// =============================================================================
// Version_Recipe - 06_MainProcess.scl
// Main process with recipe-based G-code and pre-scan validation
// =============================================================================

// -----------------------------------------------------------------------------
// FB_InputManager - OR-combine inputs from HMI, Panel, Remote
// DOC:
//  purpose: Create single rising-edge command outputs (Cmd_*) from multiple input sources.
//  inputs: HMI_*, Panel_*, Rem_* (Bool) - raw button states (level)
//  outputs: Cmd_* (Bool) - one-shot rising-edge commands for the system
//  notes: Uses prev* latches to detect rising edges; keeps logic simple for deterministic behavior.
// -----------------------------------------------------------------------------
FUNCTION_BLOCK "FB_InputManager"
{ S7_Optimized_Access := 'TRUE' }
VERSION : 1.0
    VAR_INPUT
        // Raw level inputs from various sources (HMI, physical panel, remote)
        HMI_Start : Bool;    // HMI Start button (level)
        HMI_Stop : Bool;     // HMI Stop button (level)
        HMI_Pause : Bool;    // HMI Pause button (level)
        HMI_Reset : Bool;    // HMI Reset button (level)
        Panel_Start : Bool;  // Physical panel Start
        Panel_Stop : Bool;   // Physical panel Stop
        Panel_Pause : Bool;  // Physical panel Pause
        Panel_Reset : Bool;  // Physical panel Reset
        Rem_Start : Bool;    // Remote Start (e.g. PLC network)
        Rem_Stop : Bool;     // Remote Stop
    END_VAR
    VAR_OUTPUT
        // One-shot command outputs (rising edge true for one cycle)
        Cmd_Start : Bool;
        Cmd_Stop : Bool;
        Cmd_Pause : Bool;
        Cmd_Reset : Bool;
    END_VAR
    VAR
        // Previous sampled raw values for edge detection
        prevStart : Bool;
        prevStop : Bool;
        prevPause : Bool;
        prevReset : Bool;
        // Combined raw inputs for current cycle
        rawStart : Bool;
        rawStop : Bool;
        rawPause : Bool;
        rawReset : Bool;
    END_VAR
BEGIN
    #rawStart := #HMI_Start OR #Panel_Start OR #Rem_Start;
    #rawStop := #HMI_Stop OR #Panel_Stop OR #Rem_Stop;
    #rawPause := #HMI_Pause OR #Panel_Pause;
    #rawReset := #HMI_Reset OR #Panel_Reset;
    #Cmd_Start := #rawStart AND NOT #prevStart;
    #Cmd_Stop := #rawStop AND NOT #prevStop;
    #Cmd_Pause := #rawPause AND NOT #prevPause;
    #Cmd_Reset := #rawReset AND NOT #prevReset;
    #prevStart := #rawStart; #prevStop := #rawStop; #prevPause := #rawPause; #prevReset := #rawReset;
END_FUNCTION_BLOCK

// -----------------------------------------------------------------------------
// FB_SafetyMonitor - Check E-Stop, Door, Air Pressure, Drives
// DOC:
//  purpose: Evaluate hardware safety inputs and bypass flags, produce SafeToRun/SafeToJog.
//  inputs: EStop_OK, Door_Closed, AirPressure_OK, DrivesReady and bypass flags.
//  outputs: SafeToRun (machine may start), SafeToJog (manual jog allowed), ErrorCode (if unsafe).
//  notes: Returns immediately on first fatal safety failure to minimize decision latency.
// -----------------------------------------------------------------------------
FUNCTION_BLOCK "FB_SafetyMonitor"
{ S7_Optimized_Access := 'TRUE' }
VERSION : 1.0
    VAR_INPUT
        EStop_OK : Bool;            // TRUE if E-stop circuit is OK (no emergency)
        Door_Closed : Bool;         // TRUE if safety door closed
        AirPressure_OK : Bool;      // TRUE if air pressure sufficient
        DrivesReady : Bool;         // TRUE if drives report ready
        // Bypass flags (from HMI) used only for testing; production should disable
        Bypass_EStop : Bool;
        Bypass_Door : Bool;
        Bypass_AirPressure : Bool;
        Bypass_Drives : Bool;
    END_VAR
    VAR_OUTPUT
        SafeToRun : Bool;           // TRUE => allowed to start program execution
        SafeToJog : Bool;           // TRUE => manual jogging permitted
        ErrorCode : Word;           // Non-zero if unsafe (map to DB_ErrorCodes)
    END_VAR
BEGIN
    // Runs every scan. RETURNs on first failing condition -- priority order matters.
    // EStop and Drive fault disable both SafeToRun and SafeToJog (jogging also forbidden).
    // Door and air pressure only disable SafeToRun (manual jog still permitted).
    #ErrorCode := 0;
    IF NOT #EStop_OK AND NOT #Bypass_EStop THEN
        // EMERGENCY STOP active -- all motion forbidden
        #SafeToRun := FALSE; #SafeToJog := FALSE; #ErrorCode := 16#0401;
        "DB_Diagnostic".Error_Text := 'Safety: EMERGENCY STOP active';
        RETURN;
    END_IF;
    // Drive readiness is NOT checked here.
    // In STATE_STOPPED, contactors are physically blocked (modePermit=0), so drives can never
    // report ready before starting. Blocking SafeToRun/SafeToJog here creates a deadlock.
    // Drive enable is handled automatically in STATE_STARTING (tonDriveReady timeout).
    // Drive faults while running are caught by prevDriveFaultX/Z detection → STATE_ERROR.
    #SafeToJog := TRUE;
    IF NOT #Door_Closed AND NOT #Bypass_Door THEN
        // Safety door open -- auto run forbidden, manual jog allowed
        #SafeToRun := FALSE; #ErrorCode := 16#0402;
        "DB_Diagnostic".Error_Text := 'Safety: Safety door is open';
        RETURN;
    END_IF;
    IF NOT #AirPressure_OK AND NOT #Bypass_AirPressure THEN
        // Air pressure insufficient -- pneumatic system will not operate
        #SafeToRun := FALSE; #ErrorCode := 16#0404;
        "DB_Diagnostic".Error_Text := 'Safety: Air pressure too low';
        RETURN;
    END_IF;
    #SafeToRun := TRUE;
END_FUNCTION_BLOCK

// -----------------------------------------------------------------------------
// FB_LimitMonitor - Check soft and hard limits
// DOC:
//  purpose: Validate current axis positions against configured soft limits and hardware limit switches.
//  inputs: ActualPos_X/Z, Homed_X/Z, HW limit switches.
//  outputs: LimitError (TRUE if any violation), ErrorCode (first matching error code).
//  notes: Soft limits from DB_MachineConfig are used; hardware limit switches take precedence.
//         Soft limits are only checked for a HOMED axis (Homed_X/Z = StatusBits.HomingDone):
//         before homing the TO position is meaningless (0 after restart, stale after a run),
//         so comparing it against limits would produce false trips.
// -----------------------------------------------------------------------------
FUNCTION_BLOCK "FB_LimitMonitor"
{ S7_Optimized_Access := 'TRUE' }
VERSION : 1.0
    VAR_INPUT
        ActualPos_X : Real;         // Current X position (mm)
        ActualPos_Z : Real;         // Current Z position (mm)
        Homed_X : Bool;             // X axis homed (StatusBits.HomingDone) -- soft limits checked only when TRUE
        Homed_Z : Bool;             // Z axis homed (StatusBits.HomingDone) -- soft limits checked only when TRUE
        // NC limit switches: TRUE=closed=OK, FALSE=open=limit triggered
        // Cable break also reads FALSE → fail-safe behavior
        HW_NC_X_Min : Bool;         // NC switch: X min (FALSE = limit hit)
        HW_NC_X_Max : Bool;         // NC switch: X max (FALSE = limit hit)
        HW_NC_Z_Min : Bool;         // NC switch: Z min (FALSE = limit hit)
        HW_NC_Z_Max : Bool;         // NC switch: Z max (FALSE = limit hit)
        // PNP NO proximity sensors: TRUE=target detected=entered limit zone
        // Triggered BEFORE NC switch → early warning + second safety layer
        HW_PNP_X_Min : Bool;        // PNP NO sensor: X min (TRUE = limit zone)
        HW_PNP_X_Max : Bool;        // PNP NO sensor: X max (TRUE = limit zone)
        HW_PNP_Z_Min : Bool;        // PNP NO sensor: Z min (TRUE = limit zone)
        HW_PNP_Z_Max : Bool;        // PNP NO sensor: Z max (TRUE = limit zone)
    END_VAR
    VAR_OUTPUT
        LimitError : Bool;          // TRUE if any soft/hard limit violated
        ErrorCode : Word;           // Specific error code for HMI/alarm
    END_VAR
BEGIN
    // Runs every scan. Soft limits are read from DB_MachineConfig.
    // Hardware limit switches take priority over soft limits (physical end stop).
    // ErrorCode shows the last triggered fault -- multiple can be active simultaneously.
    #LimitError := FALSE; #ErrorCode := 0;
    // --- Software (Soft) Limits ---
    // Only checked while the axis is homed: an un-homed axis has no valid position
    // reference, so soft limits cannot mean anything before the reference seek completes.
    IF #Homed_X THEN
        IF #ActualPos_X < "DB_MachineConfig".SoftLimit_MinX THEN
            #LimitError := TRUE; #ErrorCode := 16#0101;
            "DB_Diagnostic".Error_Text := 'Limit: X axis below minimum soft limit';
        END_IF;
        IF #ActualPos_X > "DB_MachineConfig".SoftLimit_MaxX THEN
            #LimitError := TRUE; #ErrorCode := 16#0102;
            "DB_Diagnostic".Error_Text := 'Limit: X axis above maximum soft limit';
        END_IF;
    END_IF;
    IF #Homed_Z THEN
        IF #ActualPos_Z < "DB_MachineConfig".SoftLimit_MinZ THEN
            #LimitError := TRUE; #ErrorCode := 16#0103;
            "DB_Diagnostic".Error_Text := 'Limit: Z axis below minimum soft limit';
        END_IF;
        IF #ActualPos_Z > "DB_MachineConfig".SoftLimit_MaxZ THEN
            #LimitError := TRUE; #ErrorCode := 16#0104;
            "DB_Diagnostic".Error_Text := 'Limit: Z axis above maximum soft limit';
        END_IF;
    END_IF;
    // --- Hardware Limit Switches ---
    // NC switches: the TO (Technology Object) is configured with these as HW limits.
    // The TO handles deceleration and stop directly -- no PLC action required.
    // Only E-Stop cuts contactor power; PLC does NOT raise LimitError on NC hits.
    //
    // PNP proximity sensors: handled separately in FB_Process (inline halt block).
    // In auto mode: PNP → MC_Halt on triggered axis + STATE_ERROR (codes 16#0121-0124).
    // In homing and manual mode: PNP is bypassed (expected zone during reference seek / manual op).
END_FUNCTION_BLOCK

// -----------------------------------------------------------------------------
// FB_AlarmManager - Unified error management and monitoring
// DOC:
//  purpose: Single place to translate error codes to text, maintain active error state,
//           append to centralized DB_Error history, and provide outputs for monitoring.
//  inputs: NewError (rising edge), NewErrorCode, AcknowledgeError (edge)
//  outputs: HasActiveError, ActiveErrorCode, ActiveErrorText, ActiveSeverity, ActiveSource, ActiveTime
//  notes: Updates legacy DB_AlarmHistory for backward compatibility but centralizes storage in DB_Error.
// -----------------------------------------------------------------------------
FUNCTION_BLOCK "FB_AlarmManager"
{ S7_Optimized_Access := 'TRUE' }
VERSION : 2.0
    VAR_INPUT
        NewError         : Bool;   // Rising edge triggers new active error
        NewErrorCode     : Word;   // Numeric code describing error
        AcknowledgeError : Bool;   // Operator ack (edge)
        ActiveProgram    : Int;    // ITEM-26: current recipe program (0=none); stored in alarm history
        ActiveLine       : Int;    // ITEM-26: current recipe line (-1=outside recipe); stored in alarm history
    END_VAR
    VAR_OUTPUT
        HasActiveError : Bool;       // TRUE while an error is active (until ack)
        ActiveErrorCode : Word;      // Current active error code
        ActiveErrorText : String[80];    // Human readable text for HMI (English)
        // ActiveErrorText_ES removed 2026-08-10 (ITEM-55 stage 1) -- Spanish error
        // text now lives in a WinCC text list keyed off DB_HMI.ErrorID.
        ActiveSeverity : Byte;       // Priority tier: 1=warning, 2=project, 3=motion/TO, 4=safety (higher preempts lower on HMI display)
        ActiveSource : String[20];   // Source category string
        ActiveTime : DTL;            // Timestamp of active error
    END_VAR
    VAR
        prevNewError : Bool;       // previous NewError for edge detection
        currentTime : DTL;         // timestamp captured at NewError
        SystemTimeStatus : Int;    // RD_SYS_T return status
        i : Int;                   // temporary loop index for history shift
        internalNewError : Bool;
        internalErrorCode : Word;
        fromQueue : Bool;           // TRUE when error came from DB_SystemEvents queue
        newHistCode   : Word;       // new error code for history push (independent of first-error latch)
        newHistText   : String[80]; // new error text for history push (independent of first-error latch)
        newHistSource : String[20]; // new error source for history push (independent of first-error latch)
        // latchedText_ES removed 2026-08-10 (ITEM-55 stage 1). It existed only to keep
        // the Spanish counterpart of the latched (displayed) error through the
        // secondary-error restore path, because DB_Error has no Details_ES field. With
        // Spanish resolved from ErrorID on the HMI there is nothing to keep in step:
        // the restore path below already puts DB_Error.Code back into ActiveErrorCode,
        // and the HMI derives the text from that.
    END_VAR
BEGIN
    #internalNewError := #NewError;
    #internalErrorCode := #NewErrorCode;
    #fromQueue := FALSE;

    // Dequeue one item per scan from DB_SystemEvents error ring buffer (written by FC_ReportError).
    // Processing one per scan is intentional: avoids two errors overwriting each other in the same
    // AlarmManager call. Any remaining items are consumed on subsequent scans.
    IF "DB_SystemEvents".EQ_Count > 0 THEN
        #internalNewError := TRUE;
        #internalErrorCode := "DB_SystemEvents".EQ_Code["DB_SystemEvents".EQ_Head];
        "DB_Diagnostic".Error_Text := "DB_SystemEvents".EQ_Details["DB_SystemEvents".EQ_Head];
        "DB_Diagnostic".Error_Code := "DB_SystemEvents".EQ_Code["DB_SystemEvents".EQ_Head];
        "DB_SystemEvents".EQ_Head  := ("DB_SystemEvents".EQ_Head + 1) MOD 4;
        "DB_SystemEvents".EQ_Count := "DB_SystemEvents".EQ_Count - 1;
        #fromQueue := TRUE;
    END_IF;

    // Handle new error
    // Queue path (fromQueue): always process — queue already guarantees one item per scan,
    //   so edge detection would drop consecutive errors when prevNewError stays TRUE.
    // Direct path (NewError input from FB_Process): edge-triggered to prevent repeated firing.
    IF #internalErrorCode <> 0 AND (#fromQueue OR (#internalNewError AND NOT #prevNewError)) THEN
        #ActiveErrorCode := #internalErrorCode;
        #SystemTimeStatus := RD_SYS_T(OUT => #currentTime);

        // Translate code -> English text.
        // Spanish was removed 2026-08-10 (ITEM-55 stage 1); the HMI resolves it from
        // DB_HMI.ErrorID via a WinCC text list. This CASE is English only, and in
        // ITEM-55 stage 2 it goes away entirely -- keep it until the WinCC text lists
        // exist, or a download leaves the operator with no error text at all.
        // Queue path: EN is overridden after the CASE with the richer diagnostic text
        //   from DB_Diagnostic.Error_Text (contains TO codes, line numbers).
        CASE #internalErrorCode OF
                // Axis Movement Errors
                16#0001: #ActiveErrorText := 'X Axis: Move command failed';
                16#0002: #ActiveErrorText := 'Z Axis: Move command failed';
                16#0003: #ActiveErrorText := 'X Axis: Homing failed';
                16#0004: #ActiveErrorText := 'Z Axis: Homing failed';
                16#0005: #ActiveErrorText := 'Drive fault - check servo';
                16#0006: #ActiveErrorText := 'Tool Axis: Move failed';
                16#0007: #ActiveErrorText := 'Tool Axis: Homing failed';
                16#0008: #ActiveErrorText := 'Motion timeout - axis stuck';
                16#0009: #ActiveErrorText := 'X drive power failed';
                16#000A: #ActiveErrorText := 'Z drive power failed';
                16#000B: #ActiveErrorText := 'Homing timeout - check ref switch';
                16#000C: #ActiveErrorText := 'Drive ready timeout - check contactor/enable wiring';
                16#000D: #ActiveErrorText := 'Tool drive power failed';           // ITEM-29
                // Raised instead of 0009/000A/000D when more than one axis reports a
                // drive-power fault in the SAME scan -- see the drive-power block in
                // FB_Process. ErrorDetail names the axes and their TO codes.
                16#000E: #ActiveErrorText := 'Drive power failed on several axes - check 24V/E-Stop';
                // EXPERIMENTAL velocity-mode path (FB_RecipeHandler STATE_VEL_WAIT). Detail
                // text says which guard fired: aborted / off path / run permission lost.
                16#000F: #ActiveErrorText := 'Velocity path fault - see detail';
                16#0012: #ActiveErrorText := 'ToolHeadLock: extend timeout - check cylinder/sensor';
                16#0010: #ActiveErrorText := 'User pressed STOP';
                // TO (Technology Object) fault poller (FB_Process, StatusBits.Error rising edge)
                16#0021: #ActiveErrorText := 'X axis TO fault - check TO diagnostics';
                16#0022: #ActiveErrorText := 'Z axis TO fault - check TO diagnostics';
                16#0023: #ActiveErrorText := 'Tool axis TO fault - check TO diagnostics';
                16#0024: #ActiveErrorText := 'Spindle TO fault - check TO diagnostics';
                // Soft Limits
                16#0101: #ActiveErrorText := 'X beyond MIN soft limit';
                16#0102: #ActiveErrorText := 'X beyond MAX soft limit';
                16#0103: #ActiveErrorText := 'Z beyond MIN soft limit';
                16#0104: #ActiveErrorText := 'Z beyond MAX soft limit';
                // PNP Proximity Zone Errors (auto mode only; homing and manual bypass these)
                16#0121: #ActiveErrorText := 'PNP zone: X axis MIN proximity';
                16#0122: #ActiveErrorText := 'PNP zone: X axis MAX proximity';
                16#0123: #ActiveErrorText := 'PNP zone: Z axis MIN proximity';
                16#0124: #ActiveErrorText := 'PNP zone: Z axis MAX proximity';
                // Tool Errors
                16#0201: #ActiveErrorText := 'Invalid tool number';
                16#0202: #ActiveErrorText := 'Tool number out of range';
                16#0203: #ActiveErrorText := 'Tool rotation timeout';
                16#0204: #ActiveErrorText := 'Retract to tool pos failed';
                16#0205: #ActiveErrorText := 'Tool rotation failed';
                16#0206: #ActiveErrorText := 'Tool change timeout - check turret drive';
                // Recipe/G-code Errors
                16#0301: #ActiveErrorText := 'Recipe: Invalid command';
                16#0302: #ActiveErrorText := 'Recipe: Parse error';
                16#0303: #ActiveErrorText := 'Recipe: Empty program';
                16#0304: #ActiveErrorText := 'Recipe: Line count zero';
                16#0305: #ActiveErrorText := 'PreScan: Path exceeds limits';
                16#0306: #ActiveErrorText := 'Recipe: Invalid feedrate';
                16#0307: #ActiveErrorText := 'Recipe: Motion timeout';
                16#0308: #ActiveErrorText := 'Recipe: Invalid tool number';
                16#0309: #ActiveErrorText := 'BackSupport cylinder error - target not reached';
                16#030A: #ActiveErrorText := 'Spindle at-speed timeout (10s)';
                16#030B: #ActiveErrorText := 'Spindle stop timeout (15s)';
                16#0310: #ActiveErrorText := 'Recipe not loaded - check TotalLines';
                16#0311: #ActiveErrorText := 'Recipe has no tool table - regenerate in CAM';
                16#0312: #ActiveErrorText := 'Recipe load from load memory failed';
                16#0313: #ActiveErrorText := 'Recipe data empty/corrupt - no END marker';
                16#0314: #ActiveErrorText := 'Recipe copy did not land - re-import recipe DB';
                16#0316: #ActiveErrorText := 'Recipe checksum mismatch - re-export and re-import';
                // Safety Errors
                16#0401: #ActiveErrorText := 'EMERGENCY STOP ACTIVE!';
                16#0402: #ActiveErrorText := 'Safety door is open';
                16#0403: #ActiveErrorText := 'Drives not ready';
                16#0404: #ActiveErrorText := 'Air pressure too low';
                16#0405: #ActiveErrorText := 'Safety interlock active';
                16#0406: #ActiveErrorText := 'E-Stop contact discrepancy!';
                // Spindle Errors
                16#0501: #ActiveErrorText := 'Spindle: Power-on failed';
                16#0502: #ActiveErrorText := 'Spindle: Run command failed';
                16#0503: #ActiveErrorText := 'Spindle: Halt failed';
                16#0504: #ActiveErrorText := 'Spindle: Speed not reached';
                16#0505: #ActiveErrorText := 'Spindle: Drive enable timeout';
                // NOTE: Siemens TO (Technology Object) error codes (16#8xxx) are NOT passed here
                // directly. They are decoded via FC_TO_ErrorText and written to
                // DB_Diagnostic.TO_ErrorText + DB_HMI.ErrorDetail at the point of failure.
                // This CASE only handles project-level error codes (16#0001-16#05FF).
                ELSE
                    #ActiveErrorText    := 'Unknown error code';
            END_CASE;
        // Queue path: override the CASE text with the detailed diagnostic text
        // (TO codes, line numbers) -- richer than the generic per-code wording.
        IF #fromQueue THEN
            #ActiveErrorText := "DB_Diagnostic".Error_Text;
        END_IF;

        // Severity & source mapping (explicit ranges)
        // Priority tiers (higher tier preempts lower on the HMI display, see latch below):
        //   4 = safety interlock (E-Stop, door, air, drives, HW limit)
        //   3 = motion / TO fault (axis, homing, drive power, soft limit, PNP zone, tool motion, spindle)
        //   2 = project error (recipe validation, tool configuration)
        //   1 = warning / info (user stop, unknown codes)
        IF #ActiveErrorCode >= 16#0400 AND #ActiveErrorCode < 16#0500 THEN
            #ActiveSeverity := 4; #ActiveSource := 'Safety';
        ELSIF #ActiveErrorCode >= 16#0111 AND #ActiveErrorCode < 16#0120 THEN
            #ActiveSeverity := 4; #ActiveSource := 'HW Limit';
        ELSIF #ActiveErrorCode >= 16#0121 AND #ActiveErrorCode < 16#0130 THEN
            #ActiveSeverity := 3; #ActiveSource := 'PNP Zone';  // PNP proximity zone errors (auto mode)
        ELSIF #ActiveErrorCode = 16#0010 THEN
            #ActiveSeverity := 1; #ActiveSource := 'Operator';  // user STOP must never preempt a real fault
        ELSIF #ActiveErrorCode >= 16#0001 AND #ActiveErrorCode <= 16#002F THEN
            #ActiveSeverity := 3; #ActiveSource := 'Axis';      // axis/homing/power, 16#0012 ToolHeadLock, 16#0021-0024 TO poller
        ELSIF #ActiveErrorCode >= 16#0101 AND #ActiveErrorCode < 16#0110 THEN
            #ActiveSeverity := 3; #ActiveSource := 'Soft Limit';
        ELSIF #ActiveErrorCode >= 16#0203 AND #ActiveErrorCode <= 16#0206 THEN
            #ActiveSeverity := 3; #ActiveSource := 'Tool';      // tool motion faults (rotation fail/timeout)
        ELSIF #ActiveErrorCode >= 16#0200 AND #ActiveErrorCode < 16#0210 THEN
            #ActiveSeverity := 2; #ActiveSource := 'Tool';      // tool configuration (invalid/out of range)
        ELSIF #ActiveErrorCode >= 16#0300 AND #ActiveErrorCode <= 16#0316 THEN
            #ActiveSeverity := 2; #ActiveSource := 'Recipe';    // <= includes 16#0310..16#0316
                                                               // (16#0315 is reserved, see TODO.md)
        ELSIF #ActiveErrorCode >= 16#0500 AND #ActiveErrorCode < 16#0510 THEN
            #ActiveSeverity := 3; #ActiveSource := 'Spindle';   // spindle motion faults
        ELSE
            #ActiveSeverity := 1; #ActiveSource := 'Unknown';
        END_IF;

        // Save new error info for history before the latch guard may restore output vars
        #newHistCode   := #ActiveErrorCode;
        #newHistText   := #ActiveErrorText;
        #newHistSource := #ActiveSource;

        // Severity-priority latch: the display (DB_Error.Code, HMI text) shows the
        // highest-severity error of the fault sequence. A new error replaces the displayed
        // one only if its priority tier is STRICTLY higher (safety 4 > motion/TO 3 >
        // project 2 > warning 1). Same or lower tier goes to history only, so the first
        // error of a tier is never pushed aside by follow-up faults of the same tier
        // (e.g. soft limit firing after the axis fault that caused it), while a TO/safety
        // fault always wins the display over a project-level error that fired first.
        // All errors always go to history. Cleared by AcknowledgeError.
        IF NOT "DB_Error".Active OR (#ActiveSeverity > "DB_Error".Severity) THEN
            #HasActiveError      := TRUE;
            #ActiveTime          := #currentTime;
            "DB_Error".Active    := TRUE;
            "DB_Error".Code      := #ActiveErrorCode;
            "DB_Error".Severity  := #ActiveSeverity;
            "DB_Error".Source    := #ActiveSource;
            IF "DB_Diagnostic".Recipe_CurrentLine >= 0 AND (#ActiveSource = 'Recipe') THEN
                "DB_Error".Line := "DB_Diagnostic".Recipe_CurrentLine;
            ELSE
                "DB_Error".Line := -1;
            END_IF;
            "DB_Error".TimeStamp := #currentTime;
            "DB_Error".Details   := #ActiveErrorText;
        ELSE
            // Same/lower-tier secondary error: restore output vars to the displayed error
            // so DB_HMI.ErrorText and callers still see the highest-priority root cause.
            // Restoring ActiveErrorCode is what keeps the HMI honest now that text is
            // resolved from the code by a WinCC text list (ITEM-55): code and text cannot
            // disagree, which is what the old latchedText_ES pairing existed to prevent.
            #ActiveErrorCode := "DB_Error".Code;
            #ActiveErrorText := "DB_Error".Details;
            #ActiveSeverity  := "DB_Error".Severity;
            #ActiveSource    := "DB_Error".Source;
            #ActiveTime      := "DB_Error".TimeStamp;
            #HasActiveError  := TRUE;
        END_IF;
        "DB_Error".TotalErrorCount := "DB_Error".TotalErrorCount + 1;
        // History: always push the new error (not the latched first-error values)
        FOR #i := 10 TO 2 BY -1 DO
            "DB_Error".History_Code[#i]    := "DB_Error".History_Code[#i - 1];
            "DB_Error".History_Time[#i]    := "DB_Error".History_Time[#i - 1];
            "DB_Error".History_Source[#i]  := "DB_Error".History_Source[#i - 1];
            "DB_Error".History_Details[#i] := "DB_Error".History_Details[#i - 1];
        END_FOR;
        "DB_Error".History_Code[1]    := #newHistCode;
        "DB_Error".History_Time[1]    := #currentTime;
        "DB_Error".History_Source[1]  := #newHistSource;
        // LEFT(..., 40): History_Details is String[40] while #newHistText is String[80].
        // Truncate explicitly rather than relying on implicit assignment truncation.
        "DB_Error".History_Details[1] := LEFT(IN := #newHistText, L := 40);
        "DB_Error".History_Index := "DB_Error".History_Index + 1;
        IF "DB_Error".History_Index > 10 THEN "DB_Error".History_Index := 1; END_IF;
        IF "DB_Error".History_Count < 10 THEN "DB_Error".History_Count := "DB_Error".History_Count + 1; END_IF;

        // ITEM-26: write to DB_AlarmHistory 20-entry ring buffer (always push new error)
        // Use #currentTime already captured above (same scan, consistent timestamp)
        IF "DB_AlarmHistory".Hist_Clear THEN
            "DB_AlarmHistory".Hist_Head   := 0;
            "DB_AlarmHistory".Hist_Count  := 0;
            "DB_AlarmHistory".Hist_SeqNum := 0;
            "DB_AlarmHistory".Hist_Clear  := FALSE;
        END_IF;
        "DB_AlarmHistory".Hist_Log["DB_AlarmHistory".Hist_Head].Timestamp  := #currentTime;
        "DB_AlarmHistory".Hist_Log["DB_AlarmHistory".Hist_Head].ErrorCode  := #newHistCode;
        "DB_AlarmHistory".Hist_Log["DB_AlarmHistory".Hist_Head].ProgramNum := #ActiveProgram;
        "DB_AlarmHistory".Hist_Log["DB_AlarmHistory".Hist_Head].LineNum    := #ActiveLine;
        "DB_AlarmHistory".Hist_Log["DB_AlarmHistory".Hist_Head].ErrorText  := LEFT(IN := #newHistText, L := 40);
        "DB_AlarmHistory".Hist_Head   := ("DB_AlarmHistory".Hist_Head + 1) MOD 20;
        "DB_AlarmHistory".Hist_SeqNum := "DB_AlarmHistory".Hist_SeqNum + 1;
        IF "DB_AlarmHistory".Hist_Count < 20 THEN
            "DB_AlarmHistory".Hist_Count := "DB_AlarmHistory".Hist_Count + 1;
        END_IF;
    END_IF;

    // Latch previous new error for edge detection
    #prevNewError := #internalNewError;

    // Acknowledge handling: clear active state but retain history snapshot
    IF #AcknowledgeError THEN
        #ActiveErrorCode := 0;
        #HasActiveError := FALSE;
        #ActiveErrorText := '';
        #ActiveSeverity := 0;
        #ActiveSource := '';
        #ActiveTime := DTL#1970-01-01-00:00:00;
        // legacy DB_AlarmHistory removed; history retained in DB_Error
        "DB_Error".Active := FALSE;
        "DB_Error".Code := 0;  // BUG FIX: clear code so DB_HMI_Errors bits go FALSE
        "DB_Error".Details := CONCAT(IN1 := "DB_Error".Details, IN2 := ' [ACK]');
    END_IF;

    // =========================================================================
    // DB_HMI_Errors - Pack error bits into Words for HMI Discrete Alarms
    // Word.Bit = one alarm line in HMI Alarm View
    // =========================================================================

    // AlarmWord_Axis: Bits 0-7
    "DB_HMI_Errors".AlarmWord_Axis :=
    BOOL_TO_WORD("DB_Error".Code = 16#0001) OR
    SHL(IN := BOOL_TO_WORD("DB_Error".Code = 16#0002), N := 1) OR
    SHL(IN := BOOL_TO_WORD("DB_Error".Code = 16#0003), N := 2) OR
    SHL(IN := BOOL_TO_WORD("DB_Error".Code = 16#0004), N := 3) OR
    SHL(IN := BOOL_TO_WORD("DB_Error".Code = 16#0005), N := 4) OR
    SHL(IN := BOOL_TO_WORD("DB_Error".Code = 16#0006), N := 5) OR
    SHL(IN := BOOL_TO_WORD("DB_Error".Code = 16#0007), N := 6) OR
    SHL(IN := BOOL_TO_WORD("DB_Error".Code = 16#0008), N := 7) OR
    SHL(IN := BOOL_TO_WORD("DB_Error".Code = 16#000D), N := 8) OR  // ITEM-29: tool drive power fault
    SHL(IN := BOOL_TO_WORD("DB_Error".Code = 16#000E), N := 9);    // multi-axis drive power fault

    // AlarmWord_Limits: Bits 0-3 soft, 4-7 hardware
    "DB_HMI_Errors".AlarmWord_Limits :=
    BOOL_TO_WORD("DB_Error".Code = 16#0101) OR
    SHL(IN := BOOL_TO_WORD("DB_Error".Code = 16#0102), N := 1) OR
    SHL(IN := BOOL_TO_WORD("DB_Error".Code = 16#0103), N := 2) OR
    SHL(IN := BOOL_TO_WORD("DB_Error".Code = 16#0104), N := 3) OR
    SHL(IN := BOOL_TO_WORD("DB_Error".Code = 16#0111), N := 4) OR
    SHL(IN := BOOL_TO_WORD("DB_Error".Code = 16#0112), N := 5) OR
    SHL(IN := BOOL_TO_WORD("DB_Error".Code = 16#0113), N := 6) OR
    SHL(IN := BOOL_TO_WORD("DB_Error".Code = 16#0114), N := 7);

    // AlarmWord_Tool: Bits 0-4
    "DB_HMI_Errors".AlarmWord_Tool :=
    BOOL_TO_WORD("DB_Error".Code = 16#0201) OR
    SHL(IN := BOOL_TO_WORD("DB_Error".Code = 16#0202), N := 1) OR
    SHL(IN := BOOL_TO_WORD("DB_Error".Code = 16#0203), N := 2) OR
    SHL(IN := BOOL_TO_WORD("DB_Error".Code = 16#0204), N := 3) OR
    SHL(IN := BOOL_TO_WORD("DB_Error".Code = 16#0205), N := 4);

    // AlarmWord_Recipe: Bits 0-7
    "DB_HMI_Errors".AlarmWord_Recipe :=
    BOOL_TO_WORD("DB_Error".Code = 16#0301) OR
    SHL(IN := BOOL_TO_WORD("DB_Error".Code = 16#0302), N := 1) OR
    SHL(IN := BOOL_TO_WORD("DB_Error".Code = 16#0303), N := 2) OR
    SHL(IN := BOOL_TO_WORD("DB_Error".Code = 16#0304), N := 3) OR
    SHL(IN := BOOL_TO_WORD("DB_Error".Code = 16#0305), N := 4) OR
    SHL(IN := BOOL_TO_WORD("DB_Error".Code = 16#0306), N := 5) OR
    SHL(IN := BOOL_TO_WORD("DB_Error".Code = 16#0307), N := 6) OR
    SHL(IN := BOOL_TO_WORD("DB_Error".Code = 16#0308), N := 7);

    // AlarmWord_Safety: Bits 0-5
    "DB_HMI_Errors".AlarmWord_Safety :=
    BOOL_TO_WORD("DB_Error".Code = 16#0401) OR
    SHL(IN := BOOL_TO_WORD("DB_Error".Code = 16#0402), N := 1) OR
    SHL(IN := BOOL_TO_WORD("DB_Error".Code = 16#0403), N := 2) OR
    SHL(IN := BOOL_TO_WORD("DB_Error".Code = 16#0404), N := 3) OR
    SHL(IN := BOOL_TO_WORD("DB_Error".Code = 16#0405), N := 4) OR
    SHL(IN := BOOL_TO_WORD("DB_Error".Code = 16#0406), N := 5);

    // AlarmWord_Spindle: Bits 0-3
    "DB_HMI_Errors".AlarmWord_Spindle :=
    BOOL_TO_WORD("DB_Error".Code = 16#0501) OR
    SHL(IN := BOOL_TO_WORD("DB_Error".Code = 16#0502), N := 1) OR
    SHL(IN := BOOL_TO_WORD("DB_Error".Code = 16#0503), N := 2) OR
    SHL(IN := BOOL_TO_WORD("DB_Error".Code = 16#0504), N := 3);

    // AlarmWord_TO: Bits 0-4
    "DB_HMI_Errors".AlarmWord_TO :=
    BOOL_TO_WORD("DB_Error".Code = 16#8401) OR
    SHL(IN := BOOL_TO_WORD("DB_Error".Code = 16#8402), N := 1) OR
    SHL(IN := BOOL_TO_WORD("DB_Error".Code = 16#8403), N := 2) OR
    SHL(IN := BOOL_TO_WORD("DB_Error".Code = 16#8404), N := 3) OR
    SHL(IN := BOOL_TO_WORD("DB_Error".Code = 16#8405), N := 4);

    // Individual Bool flags (derived from DB_Error.Code)
    "DB_HMI_Errors".Err_X_MoveFailed       := ("DB_Error".Code = 16#0001);
    "DB_HMI_Errors".Err_Z_MoveFailed       := ("DB_Error".Code = 16#0002);
    "DB_HMI_Errors".Err_X_HomingFailed     := ("DB_Error".Code = 16#0003);
    "DB_HMI_Errors".Err_Z_HomingFailed     := ("DB_Error".Code = 16#0004);
    "DB_HMI_Errors".Err_DriveFault         := ("DB_Error".Code = 16#0005);
    "DB_HMI_Errors".Err_ToolDrivePower     := ("DB_Error".Code = 16#000D);  // ITEM-29
    "DB_HMI_Errors".Err_ToolMoveFailed     := ("DB_Error".Code = 16#0006);
    "DB_HMI_Errors".Err_ToolHomingFailed   := ("DB_Error".Code = 16#0007);
    "DB_HMI_Errors".Err_MotionTimeout      := ("DB_Error".Code = 16#0008);
    "DB_HMI_Errors".Err_LockExtendTimeout  := ("DB_Error".Code = 16#0012);
    "DB_HMI_Errors".Err_SoftLimit_X_Min    := ("DB_Error".Code = 16#0101);
    "DB_HMI_Errors".Err_SoftLimit_X_Max    := ("DB_Error".Code = 16#0102);
    "DB_HMI_Errors".Err_SoftLimit_Z_Min    := ("DB_Error".Code = 16#0103);
    "DB_HMI_Errors".Err_SoftLimit_Z_Max    := ("DB_Error".Code = 16#0104);
    "DB_HMI_Errors".Err_HWLimit_X_Min      := ("DB_Error".Code = 16#0111);
    "DB_HMI_Errors".Err_HWLimit_X_Max      := ("DB_Error".Code = 16#0112);
    "DB_HMI_Errors".Err_HWLimit_Z_Min      := ("DB_Error".Code = 16#0113);
    "DB_HMI_Errors".Err_HWLimit_Z_Max      := ("DB_Error".Code = 16#0114);
    "DB_HMI_Errors".Err_InvalidToolNum     := ("DB_Error".Code = 16#0201);
    "DB_HMI_Errors".Err_ToolOutOfRange     := ("DB_Error".Code = 16#0202);
    "DB_HMI_Errors".Err_ToolRotTimeout     := ("DB_Error".Code = 16#0203);
    "DB_HMI_Errors".Err_ToolRetractFail    := ("DB_Error".Code = 16#0204);
    "DB_HMI_Errors".Err_ToolRotFailed      := ("DB_Error".Code = 16#0205);
    "DB_HMI_Errors".Err_Recipe_InvalidCmd  := ("DB_Error".Code = 16#0301);
    "DB_HMI_Errors".Err_Recipe_ParseErr    := ("DB_Error".Code = 16#0302);
    "DB_HMI_Errors".Err_Recipe_Empty       := ("DB_Error".Code = 16#0303);
    "DB_HMI_Errors".Err_Recipe_NoLines     := ("DB_Error".Code = 16#0304);
    "DB_HMI_Errors".Err_PreScan_Limits     := ("DB_Error".Code = 16#0305);
    "DB_HMI_Errors".Err_Recipe_Feedrate    := ("DB_Error".Code = 16#0306);
    "DB_HMI_Errors".Err_Recipe_Timeout     := ("DB_Error".Code = 16#0307);
    "DB_HMI_Errors".Err_Recipe_ToolNum     := ("DB_Error".Code = 16#0308);
    "DB_HMI_Errors".Err_EStop              := ("DB_Error".Code = 16#0401);
    "DB_HMI_Errors".Err_EStop_Discrepancy  := ("DB_Error".Code = 16#0406);
    "DB_HMI_Errors".Err_DoorOpen           := ("DB_Error".Code = 16#0402);
    "DB_HMI_Errors".Err_DrivesNotReady     := ("DB_Error".Code = 16#0403);
    "DB_HMI_Errors".Err_AirPressure        := ("DB_Error".Code = 16#0404);
    "DB_HMI_Errors".Err_SafetyInterlock    := ("DB_Error".Code = 16#0405);
    "DB_HMI_Errors".Err_Spindle_Power      := ("DB_Error".Code = 16#0501);
    "DB_HMI_Errors".Err_Spindle_Run        := ("DB_Error".Code = 16#0502);
    "DB_HMI_Errors".Err_Spindle_Halt       := ("DB_Error".Code = 16#0503);
    "DB_HMI_Errors".Err_Spindle_Speed      := ("DB_Error".Code = 16#0504);
    "DB_HMI_Errors".Err_TO_Position        := ("DB_Error".Code = 16#8401);
    "DB_HMI_Errors".Err_TO_Velocity        := ("DB_Error".Code = 16#8402);
    "DB_HMI_Errors".Err_TO_NotReady        := ("DB_Error".Code = 16#8403);
    "DB_HMI_Errors".Err_TO_NotEnabled      := ("DB_Error".Code = 16#8404);
    "DB_HMI_Errors".Err_TO_LimitExceeded   := ("DB_Error".Code = 16#8405);

    // Summary flags (non-zero Word = category has error)
    "DB_HMI_Errors".AnyAxisError    := ("DB_HMI_Errors".AlarmWord_Axis <> 0);
    "DB_HMI_Errors".AnyLimitError   := ("DB_HMI_Errors".AlarmWord_Limits <> 0);
    "DB_HMI_Errors".AnyToolError    := ("DB_HMI_Errors".AlarmWord_Tool <> 0);
    "DB_HMI_Errors".AnyRecipeError  := ("DB_HMI_Errors".AlarmWord_Recipe <> 0);
    "DB_HMI_Errors".AnySafetyError  := ("DB_HMI_Errors".AlarmWord_Safety <> 0);
    "DB_HMI_Errors".AnySpindleError := ("DB_HMI_Errors".AlarmWord_Spindle <> 0);
    "DB_HMI_Errors".AnyError        := "DB_Error".Active;

END_FUNCTION_BLOCK

// -----------------------------------------------------------------------------
// FB_ManualMode - Manual jog, home, move operations
// DOC:
//  purpose: Provide manual control and single-axis operations for operator (jog, absolute move, homing).
//  inputs: Enable (activation), SelectedAxis, Jog buttons, MoveAbsolute, Home commands, SafeToJog
//  outputs: Busy/Done/Error flags, AxisName/Position, ToolPosition
//  notes: Designed to be used in Manual mode only; delegates axis operations to axis FBs.
// -----------------------------------------------------------------------------
FUNCTION_BLOCK "FB_ManualMode"
{ S7_Optimized_Access := 'TRUE' }
VERSION : 1.2
    VAR_INPUT
        Enable : Bool;              // Enable manual mode (true = active)
        SelectedAxis : Int;         // 0=X,1=Z,2=Tool,3=Spindle
        Jog_Plus : Bool;            // Jog positive direction (level)
        Jog_Minus : Bool;           // Jog negative direction (level)
        JogSpeed : Real;            // Jog velocity (mm/s)
        MoveAbsolute : Bool;        // Trigger absolute move
        TargetPosition : Real;      // Absolute target position (mm)
        HomeAxis : Bool;            // Home selected axis
        HomeAll : Bool;             // Home all axes
        HomingMode : Int;           // Homing mode selection
        HomePosition : Real;        // Home position parameter (if used)
        GoSafe : Bool;              // Move to safe position
        GoZero : Bool;              // Move to zero position
        SafeToJog : Bool;           // From safety monitor
        Reset : Bool;               // Reset manual FB state
        PNP_X_Min : Bool;           // X min PNP sensor -- TRUE = in limit zone (for pre-homing clearance)
        PNP_Z_Min : Bool;           // Z min PNP sensor -- TRUE = in limit zone
        ToolStepCW : Bool;          // Tool step clockwise
        ToolStepCCW : Bool;         // Tool step counter-clockwise
        ToolStepAngle : Real;       // Angle per tool step (deg)
        ToolStepSpeed : Real;       // Velocity for tool step (deg/s)
    END_VAR
    VAR_OUTPUT
        Busy : Bool;
        Done : Bool;
        Error : Bool;
        ErrorID : Word;
        AxisName : String[10];      // Display name for selected axis
        AxisPosition : Real;        // Current axis position reported
        AxisHomed : Bool;
        AxisReady : Bool;
        ToolPosition : Real;
        ActiveAxis : Int;           // Axis currently controlled (-1 = none)
        HomingActive : Bool;        // TRUE = homing motion in progress (for limit bypass)
    END_VAR
    VAR_IN_OUT
        Axis_X : TO_PositioningAxis; // Axis technology objects (in/out interface)
        Axis_Z : TO_PositioningAxis;
        Axis_Tool : TO_PositioningAxis;
        Axis_Spindle : TO_PositioningAxis;
    END_VAR
    VAR
        state : Int;                // Local state for manual FB
        // Motion FB instances used by manual mode
        fbJogX, fbJogZ, fbJogTool : "FB_Axis_Jog";
        fbMoveX, fbMoveZ : "FB_Axis_AbsPos";
        fbMoveToolAbs : "FB_Axis_AbsPos";  // Manual > MOVE ABSOLUTE (requires homing)
        fbMoveTool : "FB_Axis_RelPos";     // Manual > TOOL STEP (does not require homing)
        fbHomeX, fbHomeZ, fbHomeTool : "FB_Axis_Home";
        // Previous input state for edge detection and one-shot triggers
        prevMoveAbs : Bool;
        prevHomeAxis : Bool;
        prevHomeAll : Bool;
        prevGoSafe : Bool;
        prevGoZero : Bool;
        prevToolStepCW : Bool;
        prevToolStepCCW : Bool;
        // Internal control flags
        bMoveX : Bool;
        bMoveZ : Bool;
        bMoveTool : Bool;
        bMoveToolAbs : Bool;
        bHomeX : Bool;
        bHomeZ : Bool;
        bHomeTool : Bool;
        bHomeAllExec : Bool;             // TRUE while HomeAll sequence is active
        homeAllStep : Int;               // HomeAll step: 1=X, 2=Z, 3=Tool
        // Homing clearance -- escape from PNP zone / move away after homing
        fbClearX : "FB_Axis_AbsPos";   // X clearance move
        fbClearZ : "FB_Axis_AbsPos";   // Z clearance hareketi
        bClearX  : Bool;               // X clearance execute flag
        bClearZ  : Bool;               // Z clearance execute flag
        bToolStepExec : Bool;
        jogAxis : Int;             // Axis selected for jogging during a jog session
        stepTarget : Real;
        moveVelocity : Real;
    END_VAR
BEGIN
    IF NOT #Enable THEN
        #state := 0; #Busy := FALSE; #Done := FALSE;
        #bMoveX := FALSE; #bMoveZ := FALSE; #bMoveTool := FALSE;
        #bHomeX := FALSE; #bHomeZ := FALSE; #bHomeTool := FALSE;
        #bHomeAllExec := FALSE; #homeAllStep := 0;
        RETURN;
    END_IF;

    IF NOT #SafeToJog THEN
        #Error := TRUE; #ErrorID := 16#0005; #state := 999;
        "DB_HMI".ErrorDetail    := 'Manual: drives not ready or E-Stop active';
    END_IF;
    IF #Reset THEN #state := 0; #Error := FALSE; #ErrorID := 0; #Done := FALSE; END_IF;

    #ToolPosition := #Axis_Tool.ActualPosition;

    CASE #SelectedAxis OF
        0: #AxisName := 'X'; #AxisPosition := #Axis_X.ActualPosition; #AxisHomed := #Axis_X.StatusBits.HomingDone; #AxisReady := #Axis_X.StatusBits.DriveReady;
        1: #AxisName := 'Z'; #AxisPosition := #Axis_Z.ActualPosition; #AxisHomed := #Axis_Z.StatusBits.HomingDone; #AxisReady := #Axis_Z.StatusBits.DriveReady;
        2: #AxisName := 'Tool'; #AxisPosition := #Axis_Tool.ActualPosition; #AxisHomed := #Axis_Tool.StatusBits.HomingDone; #AxisReady := #Axis_Tool.StatusBits.DriveReady;
        3: #AxisName := 'Spindle'; #AxisPosition := #Axis_Spindle.ActualVelocity; #AxisHomed := TRUE; #AxisReady := #Axis_Spindle.StatusBits.DriveReady;
    END_CASE;

    CASE #state OF
        0: // IDLE
            #Busy := FALSE; #Done := FALSE; #ActiveAxis := -1; #HomingActive := FALSE;
            IF (#Jog_Plus OR #Jog_Minus) AND #SafeToJog THEN #jogAxis := #SelectedAxis; #state := 10; END_IF;
            IF #MoveAbsolute AND NOT #prevMoveAbs THEN #state := 30; END_IF;
            IF #HomeAxis AND NOT #prevHomeAxis THEN #state := 40; END_IF;
            IF #HomeAll AND NOT #prevHomeAll THEN #state := 50; END_IF;
            IF #GoSafe AND NOT #prevGoSafe THEN #state := 60; END_IF;
            IF #GoZero AND NOT #prevGoZero THEN #state := 70; END_IF;
            // moveVelocity must be set here -- FB call comes at the end of the same scan;
            // if set in state 20 it arrives one scan late and MC_MoveRelative starts at 0 speed.
            IF #ToolStepCW  AND NOT #prevToolStepCW  THEN
                #stepTarget    :=  #ToolStepAngle;
                #moveVelocity  := #ToolStepSpeed;
                #bMoveTool     := TRUE;
                #state         := 20;
            END_IF;
            IF #ToolStepCCW AND NOT #prevToolStepCCW THEN
                #stepTarget    := -#ToolStepAngle;
                #moveVelocity  := #ToolStepSpeed;
                #bMoveTool     := TRUE;
                #state         := 20;
            END_IF;

        10: // JOGGING
            #Busy := TRUE; #ActiveAxis := #jogAxis;
            IF NOT #Jog_Plus AND NOT #Jog_Minus THEN #state := 99; END_IF;

        20: // TOOL STEP
            #Busy := TRUE; #ActiveAxis := 2;
            #moveVelocity := #ToolStepSpeed;
            #state := 80;

        30: // MOVE ABSOLUTE
            #Busy := TRUE;
            // Soft-limit guard: once the axis is homed, reject targets outside the
            // configured soft limits (no motion started, hint shown, back to IDLE).
            // Un-homed axes are not checked -- position is meaningless before homing
            // (AbsPos on an un-homed axis is rejected by the TO itself anyway).
            IF (#SelectedAxis = 0 AND #Axis_X.StatusBits.HomingDone
                AND (#TargetPosition < "DB_MachineConfig".SoftLimit_MinX
                     OR #TargetPosition > "DB_MachineConfig".SoftLimit_MaxX))
            OR (#SelectedAxis = 1 AND #Axis_Z.StatusBits.HomingDone
                AND (#TargetPosition < "DB_MachineConfig".SoftLimit_MinZ
                     OR #TargetPosition > "DB_MachineConfig".SoftLimit_MaxZ)) THEN
                "DB_HMI".ErrorDetail    := 'Manual: target outside soft limits - move rejected';
                #state := 0;
            ELSE
                #stepTarget := #TargetPosition; #moveVelocity := #JogSpeed;
                CASE #SelectedAxis OF
                    0: #bMoveX    := TRUE; #ActiveAxis := 0;
                    1: #bMoveZ    := TRUE; #ActiveAxis := 1;
                    2: #bMoveToolAbs := TRUE; #ActiveAxis := 2;  // AbsPos -- requires prior homing
                END_CASE;
                #state := 80;
            END_IF;

        40: // HOME AXIS INIT -- if in PNP zone, clear it first, then home
            #Busy := TRUE; #HomingActive := TRUE;
            CASE #SelectedAxis OF
                0: // X axis
                    #ActiveAxis := 0;
                    IF #PNP_X_Min THEN
                        // In X min PNP zone → clearance move first
                        #bClearX := TRUE;
                        #state := 41;
                    ELSE
                        #bHomeX := TRUE;
                        #state := 80;
                    END_IF;
                1: // Z axis
                    #ActiveAxis := 1;
                    IF #PNP_Z_Min THEN
                        #bClearZ := TRUE;
                        #state := 41;
                    ELSE
                        #bHomeZ := TRUE;
                        #state := 80;
                    END_IF;
                2: // Tool axis -- no PNP zone
                    #bHomeTool := TRUE; #ActiveAxis := 2;
                    #state := 80;
            END_CASE;

        41: // PRE-HOME CLEARANCE WAIT -- wait for clearance move out of PNP zone to finish
            #Busy := TRUE; #HomingActive := TRUE;
            IF #bClearX AND #fbClearX.Done THEN
                #bClearX := FALSE; #bHomeX := TRUE; #state := 80;
            ELSIF #bClearZ AND #fbClearZ.Done THEN
                #bClearZ := FALSE; #bHomeZ := TRUE; #state := 80;
            ELSIF (#bClearX AND #fbClearX.Error) OR (#bClearZ AND #fbClearZ.Error) THEN
                #bClearX := FALSE; #bClearZ := FALSE;
                #state := 999; #ErrorID := 16#0001;
                "DB_HMI".ErrorDetail    := 'Manual: pre-home clearance move failed';
            END_IF;

        50: // HOME ALL INIT -- clear required axes from PNP zone, then home X → Z → Tool
            #Busy := TRUE; #HomingActive := TRUE; #ActiveAxis := -1;
            #bClearX := #PNP_X_Min;   // Clearance only needed if inside PNP zone
            #bClearZ := #PNP_Z_Min;
            IF #bClearX OR #bClearZ THEN
                #state := 51;          // Clearance first
            ELSE
                #homeAllStep := 1; #bHomeX := TRUE; #bHomeAllExec := TRUE; #state := 80;
            END_IF;

        51: // HOME ALL PRE-CLEARANCE WAIT -- wait until both axes have cleared PNP zone
            #Busy := TRUE; #HomingActive := TRUE;
            IF (NOT #bClearX OR #fbClearX.Done) AND (NOT #bClearZ OR #fbClearZ.Done) THEN
                #bClearX := FALSE; #bClearZ := FALSE;
                #homeAllStep := 1; #bHomeX := TRUE; #bHomeAllExec := TRUE; #state := 80;
            ELSIF (#bClearX AND #fbClearX.Error) OR (#bClearZ AND #fbClearZ.Error) THEN
                #bClearX := FALSE; #bClearZ := FALSE;
                #state := 999; #ErrorID := 16#0001;
                "DB_HMI".ErrorDetail    := 'Manual: pre-home clearance move failed (Home All)';
            END_IF;

        60: // GO SAFE
            #Busy := TRUE; #moveVelocity := "DB_MachineConfig".RapidVelocity;
            CASE #SelectedAxis OF
                0: #bMoveX := TRUE; #stepTarget := "DB_MachineConfig".SafePos_X; #ActiveAxis := 0;
                1: #bMoveZ := TRUE; #stepTarget := "DB_MachineConfig".SafePos_Z; #ActiveAxis := 1;
            END_CASE;
            #state := 80;

        70: // GO ZERO
            #Busy := TRUE; #stepTarget := 0.0; #moveVelocity := "DB_MachineConfig".RapidVelocity;
            CASE #SelectedAxis OF
                0: #bMoveX := TRUE; #ActiveAxis := 0;
                1: #bMoveZ := TRUE; #ActiveAxis := 1;
            END_CASE;
            #state := 80;

        80: // WAIT FOR COMPLETE
            #Busy := TRUE;
            // HomingActive: set while any homing flag is still active
            #HomingActive := #bHomeX OR #bHomeZ OR #bHomeTool OR #bHomeAllExec;
            // Normal moves -- go directly to 99 on completion
            IF #bMoveX AND #fbMoveX.Done THEN #state := 99; END_IF;
            IF #bMoveX AND #fbMoveX.Error THEN
                #state := 999; #ErrorID := 16#0001;
                "DB_HMI".ErrorDetail    := CONCAT(IN1 := 'Manual X move: TO:', IN2 := "FC_TO_ErrorText"(Code := #fbMoveX.ErrorID));
            END_IF;
            IF #bMoveZ AND #fbMoveZ.Done THEN #state := 99; END_IF;
            IF #bMoveZ AND #fbMoveZ.Error THEN
                #state := 999; #ErrorID := 16#0002;
                "DB_HMI".ErrorDetail    := CONCAT(IN1 := 'Manual Z move: TO:', IN2 := "FC_TO_ErrorText"(Code := #fbMoveZ.ErrorID));
            END_IF;
            IF #bMoveTool    AND #fbMoveTool.Done    THEN #state := 99; END_IF;
            IF #bMoveTool    AND #fbMoveTool.Error   THEN
                #state := 999; #ErrorID := 16#0006;
                "DB_HMI".ErrorDetail    := CONCAT(IN1 := 'Manual tool step: TO:', IN2 := "FC_TO_ErrorText"(Code := #fbMoveTool.ErrorID));
            END_IF;
            IF #bMoveToolAbs AND #fbMoveToolAbs.Done  THEN #state := 99; END_IF;
            IF #bMoveToolAbs AND #fbMoveToolAbs.Error THEN
                #state := 999; #ErrorID := 16#0006;
                "DB_HMI".ErrorDetail    := CONCAT(IN1 := 'Manual tool abs: TO:', IN2 := "FC_TO_ErrorText"(Code := #fbMoveToolAbs.ErrorID));
            END_IF;
            // Single-axis homing -- on completion go to post-clearance (guarded: not during HomeAll)
            IF #bHomeX AND NOT #bHomeAllExec AND #fbHomeX.Done THEN
                #bHomeX := FALSE; #bClearX := TRUE; #state := 82;
            END_IF;
            IF #bHomeZ AND NOT #bHomeAllExec AND #fbHomeZ.Done THEN
                #bHomeZ := FALSE; #bClearZ := TRUE; #state := 82;
            END_IF;
            IF #bHomeTool AND NOT #bHomeAllExec AND #fbHomeTool.Done THEN #state := 99; END_IF;  // Tool axis has no PNP zone (individual home)
            IF #bHomeTool AND NOT #bHomeAllExec AND #fbHomeTool.Error THEN
                #state := 999; #ErrorID := 16#0007;
                "DB_HMI".ErrorDetail    := CONCAT(IN1 := 'Manual tool home: TO:', IN2 := "FC_TO_ErrorText"(Code := #fbHomeTool.ErrorID));
            END_IF;
            // HomeAll: sequential X → Z → Tool
            IF #bHomeAllExec THEN
                IF #homeAllStep = 1 THEN
                    // Step 1: home X
                    IF #fbHomeX.Done THEN
                        #bHomeX := FALSE; #homeAllStep := 2; #bHomeZ := TRUE;
                    ELSIF #fbHomeX.Error THEN
                        #bHomeX := FALSE; #bHomeAllExec := FALSE; #homeAllStep := 0;
                        #state := 999; #ErrorID := 16#0003;
                        "DB_HMI".ErrorDetail    := CONCAT(IN1 := 'Manual home all X: TO:', IN2 := "FC_TO_ErrorText"(Code := #fbHomeX.ErrorID));
                    END_IF;
                ELSIF #homeAllStep = 2 THEN
                    // Step 2: home Z
                    IF #fbHomeZ.Done THEN
                        #bHomeZ := FALSE;
                        IF NOT "DB_MachineConfig".Bypass_ToolAxis THEN
                            #homeAllStep := 3; #bHomeTool := TRUE;
                        ELSE
                            #bHomeAllExec := FALSE; #homeAllStep := 0;
                            #bClearX := TRUE; #bClearZ := TRUE; #state := 82;
                        END_IF;
                    ELSIF #fbHomeZ.Error THEN
                        #bHomeZ := FALSE; #bHomeAllExec := FALSE; #homeAllStep := 0;
                        #state := 999; #ErrorID := 16#0004;
                        "DB_HMI".ErrorDetail    := CONCAT(IN1 := 'Manual home all Z: TO:', IN2 := "FC_TO_ErrorText"(Code := #fbHomeZ.ErrorID));
                    END_IF;
                ELSIF #homeAllStep = 3 THEN
                    // Step 3: home Tool
                    IF #fbHomeTool.Done THEN
                        #bHomeTool := FALSE; #bHomeAllExec := FALSE; #homeAllStep := 0;
                        #bClearX := TRUE; #bClearZ := TRUE; #state := 82;
                    ELSIF #fbHomeTool.Error THEN
                        #bHomeTool := FALSE; #bHomeAllExec := FALSE; #homeAllStep := 0;
                        #state := 999; #ErrorID := 16#0007;
                        "DB_HMI".ErrorDetail    := CONCAT(IN1 := 'Manual home all Tool: TO:', IN2 := "FC_TO_ErrorText"(Code := #fbHomeTool.ErrorID));
                    END_IF;
                END_IF;
            END_IF;

        82: // POST-HOME CLEARANCE WAIT -- move away from PNP zone after homing
            #Busy := TRUE; #HomingActive := FALSE;  // Homing done, clearance move in progress
            IF (NOT #bClearX OR #fbClearX.Done) AND (NOT #bClearZ OR #fbClearZ.Done) THEN
                #bClearX := FALSE; #bClearZ := FALSE; #state := 99;
            ELSIF (#bClearX AND #fbClearX.Error) OR (#bClearZ AND #fbClearZ.Error) THEN
                #bClearX := FALSE; #bClearZ := FALSE;
                #state := 999; #ErrorID := 16#0001;
                "DB_HMI".ErrorDetail    := 'Manual: post-home clearance move failed';
            END_IF;

        99: // COMPLETE
            #Busy := FALSE; #Done := TRUE; #HomingActive := FALSE;
            #bMoveX := FALSE; #bMoveZ := FALSE; #bMoveTool := FALSE; #bMoveToolAbs := FALSE;
            #bHomeX := FALSE; #bHomeZ := FALSE; #bHomeTool := FALSE;
            #bHomeAllExec := FALSE; #homeAllStep := 0;
            #bClearX := FALSE; #bClearZ := FALSE;
            #ActiveAxis := -1;
            #state := 0;

        999: // ERROR
            #Error := TRUE; #Busy := FALSE; #HomingActive := FALSE;
            #bMoveX := FALSE; #bMoveZ := FALSE; #bMoveTool := FALSE; #bMoveToolAbs := FALSE;
            #bHomeAllExec := FALSE; #homeAllStep := 0;
            #bClearX := FALSE; #bClearZ := FALSE;
    END_CASE;

    IF #state = 0 THEN
        #prevMoveAbs := #MoveAbsolute; #prevHomeAxis := #HomeAxis; #prevHomeAll := #HomeAll;
        #prevGoSafe := #GoSafe; #prevGoZero := #GoZero;
    END_IF;

    // FB Calls
    #fbJogX(JogForward := (#Jog_Plus AND #jogAxis = 0 AND #state = 10),
            JogBackward := (#Jog_Minus AND #jogAxis = 0 AND #state = 10),
            Velocity := #JogSpeed, Axis := #Axis_X);
    #fbJogZ(JogForward := (#Jog_Plus AND #jogAxis = 1 AND #state = 10),
            JogBackward := (#Jog_Minus AND #jogAxis = 1 AND #state = 10),
            Velocity := #JogSpeed, Axis := #Axis_Z);
    #fbJogTool(JogForward  := (#Jog_Plus  AND #jogAxis = 2 AND #state = 10),
               JogBackward := (#Jog_Minus AND #jogAxis = 2 AND #state = 10),
               Velocity    := #JogSpeed, Axis := #Axis_Tool);
    #fbMoveX(Execute := #bMoveX, Position := #stepTarget, Velocity := #moveVelocity, Axis := #Axis_X);
    #fbMoveZ(Execute := #bMoveZ, Position := #stepTarget, Velocity := #moveVelocity, Axis := #Axis_Z);
    #fbMoveTool(Execute := #bMoveTool, Distance := #stepTarget, Velocity := #moveVelocity, Axis := #Axis_Tool);
    #fbMoveToolAbs(Execute := #bMoveToolAbs, Position := #stepTarget, Velocity := #moveVelocity, Axis := #Axis_Tool);
    #fbHomeX(Execute := #bHomeX, Mode := #HomingMode, Position := #HomePosition, Axis := #Axis_X);
    #fbHomeZ(Execute := #bHomeZ, Mode := #HomingMode, Position := #HomePosition, Axis := #Axis_Z);
    #fbHomeTool(Execute := #bHomeTool, Mode := #HomingMode, Position := #HomePosition, Axis := #Axis_Tool);
    // Homing clearance moves:
    //   Pre-home:  when in PNP zone, move to safe position before starting homing
    //   Post-home: move away from PNP zone after homing completes
    //   Target: HomeOffset + PostHome_Clearance (same position in both cases)
    #fbClearX(Execute  := #bClearX,
              Position := "DB_MachineConfig".HomeOffset_X + "DB_MachineConfig".PostHome_Clearance,
              Velocity := "DB_MachineConfig".HomeVelocity,
              Axis     := #Axis_X);
    #fbClearZ(Execute  := #bClearZ,
              Position := "DB_MachineConfig".HomeOffset_Z + "DB_MachineConfig".PostHome_Clearance,
              Velocity := "DB_MachineConfig".HomeVelocity,
              Axis     := #Axis_Z);
    #prevToolStepCW  := #ToolStepCW;
    #prevToolStepCCW := #ToolStepCCW;
END_FUNCTION_BLOCK

// -----------------------------------------------------------------------------
// FB_Process - Main supervisory state machine with PRE-SCAN
// -----------------------------------------------------------------------------
FUNCTION_BLOCK "FB_Process"
{ S7_Optimized_Access := 'TRUE' }
VERSION : 4.0
    VAR_INPUT Panel_Start : Bool; Panel_Stop : Bool; Panel_Pause : Bool; Panel_Reset : Bool;
              Rem_Start : Bool; Rem_Stop : Bool;
              EStop_OK : Bool := TRUE; Door_Closed : Bool := TRUE; AirPressure_OK : Bool := TRUE;
              // NC limit switches (FALSE = limit hit, fail-safe)
              HW_NC_X_Min : Bool; HW_NC_X_Max : Bool; HW_NC_Z_Min : Bool; HW_NC_Z_Max : Bool;
              // PNP NO proximity sensors (TRUE = limit zone, pre-warning before NC)
              HW_PNP_X_Min : Bool; HW_PNP_X_Max : Bool; HW_PNP_Z_Min : Bool; HW_PNP_Z_Max : Bool; END_VAR
    VAR_OUTPUT Running : Bool; IsPaused : Bool; Error : Bool; StatusID : Int; CurrentTool : Int; SafeToRun : Bool; END_VAR
    VAR_IN_OUT Axis_X : TO_PositioningAxis; Axis_Z : TO_PositioningAxis;
               Axis_Tool : TO_PositioningAxis; Axis_Spindle : TO_PositioningAxis; END_VAR
    VAR State : Int;

        // Recipe handlers -- all bound to "DB_SelectedRecipe", never to a
        // DB_RecipeProgram* (those live in load memory; see fbRecipeLoader)
        fbRecipeHandler : "FB_RecipeHandler";
        fbPreScan : "FB_RecipePreScan";
        // Load-memory recipe copy (2026-08-04): copies the selected
        // DB_RecipeProgram* into DB_SelectedRecipe in STATE_RECIPE_LOAD(11)
        fbRecipeLoader : "FB_RecipeLoader";

        // Support FBs
        fbToolChanger : "FB_ToolChanger";
        fbHomeX, fbHomeZ, fbHomeTool : "FB_Axis_Home";
        fbSpindleControl : "FB_SpindleControl";
        fbManualMode : "FB_ManualMode";
        fbPowerX, fbPowerZ, fbPowerTool : "FB_Axis_Power";
        fbResetX, fbResetZ, fbResetTool, fbResetSpindle : "FB_Axis_Reset";
        fbInputs : "FB_InputManager";
        fbLimitMonitor : "FB_LimitMonitor";
        fbSafetyMonitor : "FB_SafetyMonitor";
        fbAlarmManager : "FB_AlarmManager";
        // Additional motion FBs for moving to position 0 after stop
        fbMoveX_Stop, fbMoveZ_Stop : "FB_Axis_AbsPos";
        // Homing clearance moves (pre + post homing)
        fbMoveX_HomeClr, fbMoveZ_HomeClr : "FB_Axis_AbsPos";
        bHomeClrX, bHomeClrZ : Bool;
        // PNP proximity sensor halt: controlled stop when PNP zone entered in auto mode
        fbHaltX_PNP, fbHaltZ_PNP : "FB_Axis_Halt";
        bHaltX_PNP, bHaltZ_PNP : Bool;  // Halt execute flags (cleared when state returns to STOPPED)
        // ITEM-31: reset/startup halt — aborts any MC_Home the TO may resume after drive power-cycle or warm restart
        fbHaltX_Reset, fbHaltZ_Reset, fbHaltTool_Reset : "FB_Axis_Halt";
        bHaltAllAxes : Bool;   // Pulse: TRUE for one scan; set by bDoHardReset + first-scan startup; cleared after FB calls

        // Control flags
        bPreScanExec : Bool;
        bRecipeLoadExec : Bool; // Level: TRUE only inside STATE_RECIPE_LOAD(11).
                                // Drives fbRecipeLoader.Execute; the FB takes the
                                // rising edge, so this must go FALSE between loads.
        bResetRecipe : Bool;    // One-shot flag to reset FB_RecipeHandler
        bStartSeq, bToolExecute, bPauseActive : Bool;
        // Pause resume spin-up: on Continue from PAUSED, spindle restarts and we wait
        // SpindleResumeSpeedupTime for it to reach speed before releasing the axes to
        // return and resume. bPauseActive stays TRUE during this window so FB_RecipeHandler
        // holds at the pause-retract point (state 802).
        bResumeSpeedup   : Bool;   // TRUE while waiting for spindle to spin back up after Continue
        tonResumeSpeedup : TON;    // Spin-up wait timer (PT = DB_MachineConfig.SpindleResumeSpeedupTime)
        // Pause resume phase 1: confirm the ToolHeadLock is engaged BEFORE the spindle spins
        // back up. Set by continueEdge, cleared when the lock confirms (which arms
        // bResumeSpeedup) or when the cylinder faults (which goes to STATE_ERROR).
        bResumeLockChk   : Bool;   // TRUE while verifying ToolHeadLock on resume from PAUSED
        bStopMoveX, bStopMoveZ : Bool;       // Flags for moving to position 0 after stop
        // Sequential homing (startup): home X then Z then Tool in active mode (mode 3)
        bHomeXExec : Bool;
        bHomeZExec : Bool;
        bHomeToolExec : Bool;
        homeSeqState : Int;   // 0=idle, 1=homing X, 2=homing Z, 3=homing Tool
        activeToolReq : Int; activeToolDone : Bool;
        newErrorFlag : Bool; newErrorCode : Word;
        bSpindleStart, bSpindleStop, bDrivesEnable : Bool;
        prevAckError, prevRestart, prevContinue, ackEdge, restartEdge, continueEdge : Bool;
        prevApplyToolConfig : Bool;   // previous ApplyToolConfig button state
        applyToolEdge : Bool;         // rising edge for apply tool mapping
        prevProdReset, prevLastCycleReset, prodResetEdge, lastCycleResetEdge : Bool;
        prevSafetyError : Bool;
        prevDriveFaultX    : Bool;  // Edge detection: X drive power failure
        prevDriveFaultZ    : Bool;  // Edge detection: Z drive power failure
        prevDriveFaultTool : Bool;  // ITEM-29: edge detection: tool axis drive power failure
        prevTOFaultX       : Bool;  // Edge detection: X axis TO fault (StatusBits.Error poller)
        prevTOFaultZ       : Bool;  // Edge detection: Z axis TO fault
        prevTOFaultTool    : Bool;  // Edge detection: Tool axis TO fault
        prevTOFaultSpindle : Bool;  // Edge detection: Spindle TO fault
        // --- Sheet-load park / fast cycle mode ---
        bRequireHoming : Bool := TRUE;  // Axis reference is suspect -> next auto start MUST home.
                                        // Latched TRUE by E-Stop, STATE_ERROR and hard reset;
                                        // cleared ONLY where a homing sequence completes.
                                        // Start value TRUE so a fresh download/power-up homes.
        bRefTrusted    : Bool;  // Recomputed in STATE_STARTING: all axes homed AND NOT bRequireHoming
        clrTargetX     : Real;  // Target for fbMoveX_HomeClr -- PNP escape (state 13) or SheetLoadPos (state 16)
        clrTargetZ     : Real;  // Target for fbMoveZ_HomeClr -- PNP escape (state 13) or SheetLoadPos (state 16)
        clrVelocity    : Real;  // Velocity for the above. HomeVelocity for the slow PNP escape (13),
                                // RapidVelocity for the park move (16) -- the park can be a long
                                // travel and must not crawl at the 5 mm/s homing clearance speed.
        parkTargetX    : Real;  // Clamped SheetLoadPos_X used by the stop/park move (fbMoveX_Stop)
        parkTargetZ    : Real;  // Clamped SheetLoadPos_Z used by the stop/park move (fbMoveZ_Stop)
        bJogBlockPlus      : Bool;  // Manual soft-limit jog gate: block jog+ (recomputed every scan)
        bJogBlockMinus     : Bool;  // Manual soft-limit jog gate: block jog- (recomputed every scan)
        bToolLockEngaged   : Bool;  // ToolHeadLock is (or may be) holding the turret
        bToolAxisBlocked   : Bool;  // Manual motion on the tool axis refused because of it
        bToolStepBlocked   : Bool;  // A turret-step button is pressed while the lock is engaged.
                                    // Separate from bToolAxisBlocked because the ToolStep buttons
                                    // ignore SelectedAxis: folding them into bToolAxisBlocked would
                                    // block an X jog while the operator holds a turret-step button.
                                    // Banner only -- the refusal itself is a NOT bToolLockEngaged
                                    // term on the FB inputs.
        // ITEM-56d: blind coordinate moves (MoveAbsolute / GoSafe / GoZero) refused while halted
        // in a PNP zone. Home/HomeAll are NOT included -- homing is the escape. Level-computed
        // every scan from #State alone, like bToolAxisBlocked above, so it needs no reset path.
        bBlindMoveBlocked  : Bool;
                                    // Both recomputed every scan -- no reset path needed
        prevManualError : Bool;  // Edge detection: manual mode error
        prevMDIExec : Bool;      // Edge detection: manual MDI execute button (STATE_MANUAL)
        bMDI_Cmd40Extend : Bool; // Latch: MDI CMD=40 Param=1 holds BackSupport extended (Param=0 releases)
        // Edge detection: manual CMD=41 buttons (STATE_MANUAL). Seeded with the live
        // button state whenever the machine is outside manual, so a button left
        // latched (or an HMI that powers up with the bit set) cannot fire on entry.
        prevBtnCmd41Release : Bool;
        prevBtnCmd41AtmoOff : Bool;
        prevBtnCmd41AtmoOn  : Bool;
        // End-of-recipe BackSupport retract (operator spec 2026-08-07). On ENTRY to a
        // terminal state (STOPPED / ERROR / COMPLETE) drive Sol_B for
        // DB_MachineConfig.CylBackSupport_EndRetractTime, then drop every coil, so the
        // next recipe always starts from a known clean state regardless of how the
        // previous one ended. bBSTerminalPrev is the edge memory; it is SEEDED TRUE on
        // hard reset so power-up (which starts in STOPPED) does not fire a retract.
        bBSEndRetract   : Bool;
        bBSTerminalNow  : Bool;   // recomputed every scan (this FB has no VAR_TEMP section)
        bBSTerminalPrev : Bool;
        tonBSEndRetract : TON;
        bInitDone    : Bool;   // TRUE after first PLC scan; prevents re-triggering startup reset
        bDoHardReset : Bool;   // Pulse: set TRUE to trigger hard-reset block this scan (startup + Cmd_Reset)

        applyIndex : Int;  // Loop index for tool config apply

        // Active recipe reference
        activeProgram : Int;
        activeLineCount : Int;

        // Recipe-carried tool table (read from active recipe Header in STATE_PRE_SCAN,
        // then applied to DB_ToolConfig / DB_MachineConfig before the pre-scan runs)
        hdrProvidesToolCfg : Bool;
        hdrToolCount       : Int;
        hdrAutoCalc        : Bool;
        hdrToolCodes       : Array[1..4] of Int;
        hdrToolAngles      : Array[1..4] of Real;

        // ToolHeadLock timers
        tonLockWait : TON;      // Fallback timeout for states 17 and 29 (T#3S)
        tonLockPreDelay : TON;  // Pre-delay before commanding extend in state 17 (T#1S)
        // TRUE = LOCK_RETRACT_WAIT exits to STATE_STOPPED (axes already parked at SheetLoadPos by STOPPING)
        // FALSE = exits to STATE_TOOL_CHANGE
        bLockAfterHoming : Bool;
        // Sheet wait (STATE_SHEET_WAIT = 14)
        bSheetWaitPhase2          : Bool;   // Phase 2: MandrelLock extending (T#5S)
        bSheetWaitPhase3          : Bool;   // Phase 3: SheetHolder retracting (T#5S)
        tonMandrelWait            : TON;    // T#5S open-loop stroke wait for MandrelLock (phase 2)
        tonSheetHolderRetract     : TON;    // T#5S open-loop wait for SheetHolder retract (phase 3)
        bMandrelRetractPulse      : Bool;   // One-shot: pulse Cmd_Retract for one scan to release MandrelLock FB from State 3
        bMandrelRetractPending    : Bool;   // ITEM-32: deferred retract — unsafe paths (Reset/Error/Complete) set this; SpindleStopSafeTime timer promotes to pulse
        tonMandrelRetractWait     : TON;    // ITEM-32: safety gate timer for deferred retract (PT = DB_MachineConfig.SpindleStopSafeTime)
        // SheetHolder is a 5/3 blocked centre (ValveType=2) -- no spring. Cmd_Retract must be
        // HELD for the whole stroke, not pulsed: a one-scan pulse energises Sol_B for one scan
        // and the blocked centre then locks the piston mid-stroke. Held for exactly
        // CylSheetHolder_RetractTime (tonSheetHolderHold below), then dropped so BOTH coils
        // de-energise and the blocked centre holds the piston -- ITEM-46. Also cleared on
        // STATE_SHEET_WAIT Ph1 so an extend always wins.
        bSheetHolderRetractHold   : Bool;   // Held: drives Cmd_Retract for the retract window only
        // ITEM-46: bounds the retract coil. Runs whenever the latch is held AND the coils can
        // actually move the piston (E-Stop OK) -- an E-Stop during the stroke pauses the window
        // instead of burning it, so the retract finishes when the E-Stop is released.
        tonSheetHolderHold        : TON;    // PT = DB_MachineConfig.CylSheetHolder_RetractTime
        bWaitingSpindleStop       : Bool;   // TRUE while STATE_STOPPING waits for spindle decel before retracting MandrelLock
        tonSpindleStopWait        : TON;    // Proportional wait before MandrelLock retract (see SpindleStopSafeTime). Fires immediately if speed was 0.
        capturedSpindleRPM        : Real;   // Speed captured when bWaitingSpindleStop is set (ITEM-28)
        spindleStopPT             : Time;   // Proportional PT for tonSpindleStopWait (ITEM-28)

        // Cycle timer
        tonElapsed : TON;
        // Homing timeout: fires if STATE_HOMING sequence takes longer than 120s
        tonHomingTimeout : TON;
        // ITEM-30: independent timeout for STATE_STOP_GOHOME (was sharing tonHomingTimeout — risky if
        // a normal homing cycle consumed most of the budget, leaving too little time for post-stop homing)
        tonStopHomeTimeout : TON;
        // Drive ready timeout: fires if drives do not become ready within 3s of STATE_STARTING
        tonDriveReady : TON;
        // Spindle deceleration wait
        tonSpindleDecel      : TON;   // Decel wait timer
        bSpindleDecelWait    : Bool;  // TRUE while waiting for decel to complete
        bSpindlePendingStart : Bool;  // Deferred start captured during decel wait
        pendingSpindleSpeed  : Real;  // Speed to apply when timer expires
        // End-of-program sanding dwell (2026-08-29). Armed at the RUNNING -> COMPLETE
        // transition, run inside STATE_COMPLETE(100). See DB_MachineConfig.SandTime_s.
        bSandActive          : Bool;  // TRUE while the sanding dwell is running
        tonSandDwell         : TON;   // Dwell timer (PT = #sandTimePT)
        sandSpeedClamped     : Real;  // SandSpeed clamped to DB_Spindle.MinSpeed/MaxSpeed
        sandTimeSec          : Int;   // SandTime_s clamped to 0..SAND_TIME_MAX_S
        sandTimePT           : Time;  // #sandTimeSec converted to a Time for tonSandDwell
        elapsedAccum : Time;         // Accumulated elapsed time
        timerRunning : Bool;         // Timer active flag
        elapsedSeconds : DInt;       // Seconds counter

        // Warm restart
        savedLineIndex : Int := -1;  // Saved line for restart (-1 = none)
        savedProgram : Int := -1;    // Saved program for restart

        // Production logging
        prevState : Int;             // For state edge detection
        prodTimeNow : DTL;
        prodTimeStatus : Int;

        // Spindle history ring buffer: previous values for change detection
        // A new snapshot is pushed only when one of these changes.
        prevSnap_State       : Int;
        prevSnap_PrevStart   : Bool;
        prevSnap_ReqStart    : Bool;
        prevSnap_StartEdge   : Bool;
        prevSnap_MoveVelBusy : Bool;  // MC_MoveVelocity.Busy -- triggers snapshot when TO accepts/drops command

    END_VAR

    CONST
        STATE_STOPPED : Int := 0;
        STATE_MANUAL : Int := 5;
        STATE_STARTING : Int := 10;
        // Copies the selected recipe out of load memory into DB_SelectedRecipe.
        // Runs BEFORE the pre-scan -- the pre-scan is what reads the lines and
        // applies the header tool table, so the buffer must be filled first.
        STATE_RECIPE_LOAD : Int := 11;
        STATE_PRE_SCAN : Int := 12;
        STATE_PRE_HOME_CLR : Int := 13;      // Pre-homing clearance move out of PNP zone
        STATE_SHEET_WAIT   : Int := 14;      // Sheet insertion: Ph1=SheetHolder extends+prompt, Ph2=MandrelLock T#5S, Ph3=SheetHolder retract T#5S → LOCK_EXTEND_WAIT
        STATE_HOMING : Int := 15;
        STATE_POST_HOME_CLR : Int := 16;     // Post-homing clearance move away from PNP zone
        STATE_STOPPING : Int := 18;
        STATE_STOP_GOHOME : Int := 19;
        STATE_STOP_GOTOZERO : Int := 21;
        STATE_PNP_HALT : Int := 22;          // PNP limit zone -- halt active, reverse jog allowed
        STATE_RUNNING : Int := 20;
        STATE_PAUSED : Int := 25;
        STATE_TOOL_CHANGE : Int := 30;
        STATE_TOOL_WAIT : Int := 35;
        STATE_LOCK_EXTEND_WAIT : Int := 17;   // ToolHeadLock engaging before RUNNING
        STATE_LOCK_RETRACT_WAIT : Int := 29;  // ToolHeadLock releasing before tool change or homing
        STATE_ERROR : Int := 999;
        // End-of-program sanding dwell (2026-08-29): upper bound on the operator-typed
        // DB_MachineConfig.SandTime_s. 600 s = 10 minutes, far beyond any real sanding
        // job, and it stops a slipped decimal or a stray keypress from leaving the
        // spindle turning unattended for hours. The clamp is the reason the config value
        // can safely be a plain Int the operator types into.
        SAND_TIME_MAX_S : Int := 600;
    END_CONST
BEGIN
    // Update HMI displays
    "DB_HMI".ActualX := #Axis_X.ActualPosition;
    "DB_HMI".ActualZ := #Axis_Z.ActualPosition;
    "DB_HMI".MachineState := #State;

    // =========================================================================
    // FIRST-SCAN STARTUP INIT
    // =========================================================================
    // On the very first PLC scan after power-up or warm restart, trigger a hard
    // reset. This forces a known-clean machine state explicitly rather than
    // relying solely on NON_RETAIN default values. Covers any case where the
    // state machine variable did not reset cleanly (e.g. mid-homing on restart).
    IF NOT #bInitDone THEN
        #bDoHardReset := TRUE;
        #bHaltAllAxes := TRUE;   // ITEM-31: abort any MC_Home the TO may auto-resume on power-up
        // Power-up ALWAYS requires homing. Set explicitly here rather than relying on the
        // hard-reset block: that block now decides from the pre-reset #State, which is 0
        // (STOPPED) on the first scan and would therefore skip the latch. The VAR default is
        // also TRUE, but only because the instance DB is NON_RETAIN -- do not depend on that.
        #bRequireHoming := TRUE;
        // BackSupport end-of-recipe retract (ITEM-41): seed the terminal-state edge memory TRUE
        // so power-up does NOT fire a retract nobody asked for. This scan ends in STOPPED (a
        // terminal state) and an unseeded edge memory would read that as a fresh entry.
        //
        // This seeding belongs HERE and nowhere else. In the general hard-reset block it would
        // also suppress the retract on an operator Reset pressed from RUNNING -- that reset sets
        // State := STOPPED, so a pre-seeded edge memory sees terminal->terminal and the cylinder
        // is left frozen mid-recipe, which is the ITEM-48 failure all over again.
        #bBSTerminalPrev := TRUE;
        #bBSEndRetract   := FALSE;
        #tonBSEndRetract(IN := FALSE, PT := "DB_MachineConfig".CylBackSupport_EndRetractTime);
        "DB_Cylinder_BackSupport".Cmd_Retract := FALSE;
        #bInitDone    := TRUE;
    END_IF;

    // Edge detection for buttons
    #ackEdge := "DB_HMI".Btn_AckError AND NOT #prevAckError;
    #prevAckError := "DB_HMI".Btn_AckError;
    #restartEdge := "DB_HMI".Btn_Restart AND NOT #prevRestart;
    #prevRestart := "DB_HMI".Btn_Restart;
    #continueEdge := "DB_HMI".Btn_Continue AND NOT #prevContinue;
    #prevContinue := "DB_HMI".Btn_Continue;
    // Apply Tool Config edge
    #applyToolEdge := "DB_HMI".Btn_ApplyToolConfig AND NOT #prevApplyToolConfig;
    #prevApplyToolConfig := "DB_HMI".Btn_ApplyToolConfig;
    #prodResetEdge := "DB_HMI".Btn_ProdReset AND NOT #prevProdReset;
    #prevProdReset := "DB_HMI".Btn_ProdReset;
    #lastCycleResetEdge := "DB_HMI".Btn_LastCycleReset AND NOT #prevLastCycleReset;
    #prevLastCycleReset := "DB_HMI".Btn_LastCycleReset;

    // Get active program from HMI (lock during RUNNING to prevent mid-program switch)
    IF #State < STATE_STARTING OR #State >= STATE_ERROR THEN
        #activeProgram := "DB_HMI".ProductSelect;
        IF #activeProgram < 1 THEN #activeProgram := 1; END_IF;
        // <<< GENERATED:PROGRAM_CLAMP -- do not hand-edit; run tools/gen_recipe_slots.py >>>
        IF #activeProgram > 10 THEN #activeProgram := 10; END_IF;  // 10 recipe slots
        // <<< END GENERATED:PROGRAM_CLAMP >>>
    END_IF;

    // Tool-slot mapping is now CAM-authored: the active recipe Header supplies the
    // tool table and it is applied on Start (STATE_PRE_SCAN). "Recipe always wins" --
    // the HMI Apply path is intentionally disabled and DB_HMI.ToolSlotCode is a
    // read-only mirror of the active mapping for display only. #applyToolEdge is still
    // computed above (harmless) but no longer copies into DB_ToolConfig.
    // (See CAM_TOOL_TABLE_HANDOVER.md.)
    FOR #applyIndex := 1 TO 4 DO
        "DB_HMI".ToolSlotCode[#applyIndex] := "DB_ToolConfig".ToolCode_List[#applyIndex];
    END_FOR;

    // Safety monitor
    #fbSafetyMonitor(EStop_OK := #EStop_OK, Door_Closed := #Door_Closed, AirPressure_OK := #AirPressure_OK,
                     DrivesReady := #fbPowerX.Status AND #fbPowerZ.Status,
                     Bypass_EStop := "DB_HMI".Bypass_EStop,
                     Bypass_Door := "DB_HMI".Bypass_Door,
                     Bypass_AirPressure := "DB_HMI".Bypass_AirPressure,
                     Bypass_Drives := "DB_HMI".Bypass_Drives);

    // Power control
    #bDrivesEnable := (#EStop_OK OR "DB_HMI".Bypass_EStop) AND (#State <> STATE_ERROR);
    #fbPowerX(Enable := #bDrivesEnable, Axis := #Axis_X);
    #fbPowerZ(Enable := #bDrivesEnable, Axis := #Axis_Z);
    #fbPowerTool(Enable := #bDrivesEnable AND NOT "DB_MachineConfig".Bypass_ToolAxis, Axis := #Axis_Tool);

    // Drive power failure detection -- capture TO ErrorID and write to diagnostic
    // Checked every scan; alarm is raised only when a new error occurs (rising edge).
    // STATE_RECIPE_LOAD(11) and STATE_PRE_SCAN(12) are treated like STATE_STOPPED(0):
    // contactors are still open during the recipe copy and
    // pre-scan (closed only in STATE_STARTING), so a drive fault here is typically a latched
    // fault from a previous run or a transient after TO reset -- not a new startup failure.
    // The drive ready check (tonDriveReady) and MC_Home.Error in STATE_STARTING handle genuine
    // startup faults. Firing STATE_ERROR in PRE_SCAN would abort the recipe validation for no reason.
    //
    // NAMING (2026-08-17): this used to be three independent blocks, one per axis, each
    // writing the SINGLE #newErrorFlag/#newErrorCode pair that FB_AlarmManager consumes
    // once per scan. X wrote 16#0009, Z overwrote it with 16#000A, Tool overwrote that
    // with 16#000D -- so a fault that hit more than one axis in the same scan ALWAYS
    // came out as "Tool drive power failed", whatever actually happened, and the two
    // earlier codes were lost entirely (no history entry, because only one NewError
    // edge ever reached the alarm manager). Field evidence 2026-08-17: X and Z both
    // latched Power_*_ErrorID = 16#8007 while DB_Error held one single 16#000D and
    // TotalErrorCount = 1.
    //
    // Now: per-axis ErrorID latching stays per-axis, but the ALARM is chosen once, from
    // what is actually in fault this scan. Exactly one axis -> that axis's own code.
    // More than one -> 16#000E, because no single axis name would be true and
    // "several drives at once" is the diagnostically useful message (shared 24 V,
    // contactor circuit, E-Stop, or the TOs still starting up).
    // Do not split this back into per-axis blocks while #newErrorCode is a single
    // variable -- that is the bug.

    // Per-axis latches: independent of which alarm gets reported, so all three survive
    // even when only one of them is the headline. Never cleared -- non-zero means that
    // axis faulted at some point this power cycle. Power_Tool_ErrorID added 2026-08-17;
    // before that the tool's code was recoverable only from the volatile FB output,
    // which Reset erases.
    IF #fbPowerX.Error THEN
        "DB_Diagnostic".Power_X_ErrorID := #fbPowerX.ErrorID;
    END_IF;
    IF #fbPowerZ.Error THEN
        "DB_Diagnostic".Power_Z_ErrorID := #fbPowerZ.ErrorID;
    END_IF;
    IF #fbPowerTool.Error THEN
        "DB_Diagnostic".Power_Tool_ErrorID := #fbPowerTool.ErrorID;
    END_IF;

    // One alarm per scan, on the rising edge of ANY of the three.
    IF (#fbPowerX.Error AND NOT #prevDriveFaultX)
       OR (#fbPowerZ.Error AND NOT #prevDriveFaultZ)
       OR (#fbPowerTool.Error AND NOT #prevDriveFaultTool) THEN

        // Fault trail: name every axis in drive-power fault right now, with its TO code.
        // A common-mode event is then visible as such even if the headline code is read
        // in isolation later. Built one CONCAT at a time, and TO_ErrorText is used as the
        // scratch for each FC result -- both deliberate, to keep every construct here
        // identical to ones already used elsewhere in this file. TO_ErrorText is given
        // its final, authoritative value in the headline block below.
        "DB_Diagnostic".Error_Text := 'DrivePower:';
        IF #fbPowerX.Error THEN
            "DB_Diagnostic".TO_ErrorText := "FC_TO_ErrorText"(Code := #fbPowerX.ErrorID);
            "DB_Diagnostic".Error_Text := CONCAT(IN1 := "DB_Diagnostic".Error_Text, IN2 := ' X=');
            "DB_Diagnostic".Error_Text := CONCAT(IN1 := "DB_Diagnostic".Error_Text, IN2 := "DB_Diagnostic".TO_ErrorText);
        END_IF;
        IF #fbPowerZ.Error THEN
            "DB_Diagnostic".TO_ErrorText := "FC_TO_ErrorText"(Code := #fbPowerZ.ErrorID);
            "DB_Diagnostic".Error_Text := CONCAT(IN1 := "DB_Diagnostic".Error_Text, IN2 := ' Z=');
            "DB_Diagnostic".Error_Text := CONCAT(IN1 := "DB_Diagnostic".Error_Text, IN2 := "DB_Diagnostic".TO_ErrorText);
        END_IF;
        IF #fbPowerTool.Error THEN
            "DB_Diagnostic".TO_ErrorText := "FC_TO_ErrorText"(Code := #fbPowerTool.ErrorID);
            "DB_Diagnostic".Error_Text := CONCAT(IN1 := "DB_Diagnostic".Error_Text, IN2 := ' Tool=');
            "DB_Diagnostic".Error_Text := CONCAT(IN1 := "DB_Diagnostic".Error_Text, IN2 := "DB_Diagnostic".TO_ErrorText);
        END_IF;

        // Headline code: single axis -> that axis. Two or three -> 16#000E.
        #newErrorFlag := TRUE;
        IF #fbPowerX.Error AND NOT #fbPowerZ.Error AND NOT #fbPowerTool.Error THEN
            #newErrorCode := 16#0009;
            "DB_Diagnostic".TO_ErrorText := "FC_TO_ErrorText"(Code := #fbPowerX.ErrorID);
        ELSIF #fbPowerZ.Error AND NOT #fbPowerX.Error AND NOT #fbPowerTool.Error THEN
            #newErrorCode := 16#000A;
            "DB_Diagnostic".TO_ErrorText := "FC_TO_ErrorText"(Code := #fbPowerZ.ErrorID);
        ELSIF #fbPowerTool.Error AND NOT #fbPowerX.Error AND NOT #fbPowerZ.Error THEN
            #newErrorCode := 16#000D;
            "DB_Diagnostic".TO_ErrorText := "FC_TO_ErrorText"(Code := #fbPowerTool.ErrorID);
        ELSE
            // Unreachable with none in fault: the edge above guarantees at least one.
            #newErrorCode := 16#000E;
            "DB_Diagnostic".TO_ErrorText := 'MultiAxis';
        END_IF;

        "DB_HMI".ErrorDetail := "DB_Diagnostic".Error_Text;

        IF #State <> STATE_ERROR AND #State <> 0 AND #State <> STATE_PRE_SCAN
           AND #State <> STATE_RECIPE_LOAD THEN
            #State := STATE_ERROR;
        END_IF;
    END_IF;

    // Edge memories: updated every scan, after the alarm decision has read them.
    #prevDriveFaultX    := #fbPowerX.Error;
    #prevDriveFaultZ    := #fbPowerZ.Error;
    #prevDriveFaultTool := #fbPowerTool.Error;

    // =========================================================================
    // TO (Technology Object) FAULT POLLER
    // =========================================================================
    // Guarantees axis TO errors ALWAYS reach the HMI. The MC_ wrapper FBs only report
    // an ErrorID while their own command is active; a TO fault outside an active command
    // (following error, TO-internal soft-limit trip, encoder/drive fault at rest) was
    // previously visible only on the TIA Portal TO diagnostics page.
    // Polls <axis>.StatusBits.Error every scan, raises a motion-tier alarm on the rising
    // edge. Skipped while the matching MC_Power FB reports a fault (the drive-power blocks
    // above already raise the more specific 16#0009/16#000A/16#000D) and while E-Stop is
    // active (the safety tier owns that case; power removal marks every axis in error).
    // TO errors are cleared by the MC_Reset calls on AckError/Reset (fbResetX/Z/Tool/Spindle).
    IF #Axis_X.StatusBits.Error AND NOT #fbPowerX.Error AND #EStop_OK THEN
        IF NOT #prevTOFaultX THEN
            #newErrorFlag := TRUE; #newErrorCode := 16#0021;
            "DB_Diagnostic".Error_Text := 'TO fault: X axis (StatusBits.Error) - check TO diagnostics';
            "DB_HMI".ErrorDetail    := 'X axis technology object fault - press Ack/Reset to clear';
            IF #State <> STATE_ERROR AND #State <> 0 AND #State <> STATE_PRE_SCAN
               AND #State <> STATE_RECIPE_LOAD THEN
                #State := STATE_ERROR;
            END_IF;
        END_IF;
        #prevTOFaultX := TRUE;
    ELSE
        #prevTOFaultX := FALSE;
    END_IF;

    IF #Axis_Z.StatusBits.Error AND NOT #fbPowerZ.Error AND #EStop_OK THEN
        IF NOT #prevTOFaultZ THEN
            #newErrorFlag := TRUE; #newErrorCode := 16#0022;
            "DB_Diagnostic".Error_Text := 'TO fault: Z axis (StatusBits.Error) - check TO diagnostics';
            "DB_HMI".ErrorDetail    := 'Z axis technology object fault - press Ack/Reset to clear';
            IF #State <> STATE_ERROR AND #State <> 0 AND #State <> STATE_PRE_SCAN
               AND #State <> STATE_RECIPE_LOAD THEN
                #State := STATE_ERROR;
            END_IF;
        END_IF;
        #prevTOFaultZ := TRUE;
    ELSE
        #prevTOFaultZ := FALSE;
    END_IF;

    IF #Axis_Tool.StatusBits.Error AND NOT #fbPowerTool.Error AND #EStop_OK
       AND NOT "DB_MachineConfig".Bypass_ToolAxis THEN
        IF NOT #prevTOFaultTool THEN
            #newErrorFlag := TRUE; #newErrorCode := 16#0023;
            "DB_Diagnostic".Error_Text := 'TO fault: Tool axis (StatusBits.Error) - check TO diagnostics';
            "DB_HMI".ErrorDetail    := 'Tool axis technology object fault - press Ack/Reset to clear';
            IF #State <> STATE_ERROR AND #State <> 0 AND #State <> STATE_PRE_SCAN
               AND #State <> STATE_RECIPE_LOAD THEN
                #State := STATE_ERROR;
            END_IF;
        END_IF;
        #prevTOFaultTool := TRUE;
    ELSE
        #prevTOFaultTool := FALSE;
    END_IF;

    // Spindle: MC_Power lives inside fbSpindleControl (no fbPowerSpindle guard here).
    // A same-scan specific spindle error (16#05xx) from FB_SpindleControl wins the display
    // anyway (same tier, first-in latch); this poller is the safety net for faults at rest.
    IF #Axis_Spindle.StatusBits.Error AND #EStop_OK THEN
        IF NOT #prevTOFaultSpindle THEN
            #newErrorFlag := TRUE; #newErrorCode := 16#0024;
            "DB_Diagnostic".Error_Text := 'TO fault: Spindle (StatusBits.Error) - check TO diagnostics';
            "DB_HMI".ErrorDetail    := 'Spindle technology object fault - press Ack/Reset to clear';
            IF #State <> STATE_ERROR AND #State <> 0 AND #State <> STATE_PRE_SCAN
               AND #State <> STATE_RECIPE_LOAD THEN
                #State := STATE_ERROR;
            END_IF;
        END_IF;
        #prevTOFaultSpindle := TRUE;
    ELSE
        #prevTOFaultSpindle := FALSE;
    END_IF;

    // Limit monitor
    #fbLimitMonitor(ActualPos_X := #Axis_X.ActualPosition, ActualPos_Z := #Axis_Z.ActualPosition,
                    Homed_X := #Axis_X.StatusBits.HomingDone, Homed_Z := #Axis_Z.StatusBits.HomingDone,
                    HW_NC_X_Min := #HW_NC_X_Min, HW_NC_X_Max := #HW_NC_X_Max,
                    HW_NC_Z_Min := #HW_NC_Z_Min, HW_NC_Z_Max := #HW_NC_Z_Max,
                    HW_PNP_X_Min := #HW_PNP_X_Min, HW_PNP_X_Max := #HW_PNP_X_Max,
                    HW_PNP_Z_Min := #HW_PNP_Z_Min, HW_PNP_Z_Max := #HW_PNP_Z_Max);
    // NOTE: FB_LimitMonitor itself now checks soft limits only for HOMED axes
    // (Homed_X/Z inputs = StatusBits.HomingDone) -- an un-homed axis can never trip a
    // soft limit. The state bypasses below remain as defense in depth:
    // During homing the axis may move outside soft limits (moving toward home switch).
    // All four homing-related states are bypassed: PRE_HOME_CLR, HOMING, POST_HOME_CLR,
    // and STOP_GOHOME. Without bypassing PRE/POST_HOME_CLR the clearance moves could
    // trip a spurious soft-limit fault before homing even begins (TO position = 0 after restart).
    // STATE_MANUAL and STATE_PNP_HALT are also bypassed: manual mode enforces soft limits
    // via directional jog gating + MoveAbsolute target rejection (never faults, so the
    // operator can always jog back into range).
    // STATE_PRE_SCAN(12) and STATE_STARTING(10) are bypassed because:
    //   RECIPE_LOAD: pure data copy out of load memory, no motion at all.
    //   PRE_SCAN: pure software validation, no motion -- TO position may be stale from last run.
    //   STARTING: contactors just closing, drives not yet ready -- homing will establish real position.
    // HW limit switch faults are caught by TO → MC_Home.Error → handled in state machine.
    IF #State = STATE_HOMING OR #State = STATE_STOP_GOHOME
       OR #State = STATE_PRE_HOME_CLR OR #State = STATE_POST_HOME_CLR
       OR #State = STATE_MANUAL OR #State = STATE_PNP_HALT
       OR #State = STATE_PRE_SCAN OR #State = STATE_STARTING
       OR #State = STATE_RECIPE_LOAD THEN
        #SafeToRun := #fbSafetyMonitor.SafeToRun;   // Soft limit bypass
    ELSE
        #SafeToRun := #fbSafetyMonitor.SafeToRun AND NOT #fbLimitMonitor.LimitError;
    END_IF;

    // Safety error handling
    // NOTE: Alarm is only raised from active states such as RUNNING/MANUAL.
    // No new alarm is raised in STOPPED (0) or ERROR (999) state;
    // this prevents drive enable delay after ACK/Reset from creating spurious alarms.
    IF NOT #fbSafetyMonitor.SafeToRun AND #fbSafetyMonitor.ErrorCode <> 0 THEN
        IF NOT #prevSafetyError AND #State <> 0 AND #State <> STATE_ERROR THEN
            #newErrorFlag := TRUE; #newErrorCode := #fbSafetyMonitor.ErrorCode;
        END_IF;
        IF #State <> 0 AND #State <> STATE_ERROR THEN #State := STATE_ERROR; END_IF;
        #prevSafetyError := TRUE;
    ELSE
        #prevSafetyError := FALSE;
    END_IF;

    // Soft limit error handling -- triggers STATE_ERROR when axis exceeds configured soft limits.
    // Un-homed axes never trip (FB_LimitMonitor Homed_X/Z gating -- position is meaningless
    // before the reference seek completes).
    // NC hardware limit switches are removed from LimitMonitor; TO handles them natively.
    // Bypassed in all four homing-related states: during homing the axis may legitimately
    // travel outside the configured limits while seeking the reference switch.
    // STATE_MANUAL and STATE_PNP_HALT also bypassed: manual mode enforces soft limits via
    // directional jog gating + MoveAbsolute target rejection instead of faulting.
    // STATE_RECIPE_LOAD(11), STATE_PRE_SCAN(12) and STATE_STARTING(10) bypassed: TO position may be stale
    // from the previous run; firing here would abort startup for a position that was valid last run.
    IF #fbLimitMonitor.LimitError AND #fbLimitMonitor.ErrorCode <> 0
       AND #State <> STATE_HOMING AND #State <> STATE_STOP_GOHOME
       AND #State <> STATE_PRE_HOME_CLR AND #State <> STATE_POST_HOME_CLR
       AND #State <> STATE_MANUAL AND #State <> STATE_PNP_HALT
       AND #State <> STATE_PRE_SCAN AND #State <> STATE_STARTING
       AND #State <> STATE_RECIPE_LOAD
       AND #State <> STATE_STOPPED AND #State <> STATE_ERROR THEN
        #newErrorFlag := TRUE;
        #newErrorCode := #fbLimitMonitor.ErrorCode;
        #State := STATE_ERROR;
    END_IF;

    // PNP proximity sensor halt -- auto mode only.
    // Bypassed in: homing states (PNP zone expected during reference seek),
    //              manual mode (operator in direct control, TO handles HW limits),
    //              STOPPED, PNP_HALT, and ERROR (no active motion to halt),
    //              STARTING / RECIPE_LOAD / PRE_SCAN (see below -- added 2026-08-16).
    // Triggers: MC_Halt on affected axis + STATE_PNP_HALT.
    // In STATE_PNP_HALT: drives stay ON, FB_ManualMode active, reverse jog allowed to escape zone.
    //
    // STARTING(10) / RECIPE_LOAD(11) / PRE_SCAN(12) added 2026-08-16 -- this is what makes the
    // documented recovery actually work. Recovery is: PNP trips -> PNP_HALT -> operator presses
    // Reset -> error acknowledged, State := STOPPED, bRequireHoming latched TRUE -> operator
    // presses Start -> homing runs and drives the axis out of the zone (the TO is configured to
    // reverse at the hardware limit, so the seek recovers from either side).
    //
    // It could never get there. STATE_STOPPED force-clears bHaltX/Z_PNP every scan, and the
    // sensor is of course still TRUE -- the axis has not moved. Start puts the machine in
    // RECIPE_LOAD(11), which was NOT bypassed, so the very first scan re-fired 16#0121 and threw
    // it straight back into PNP_HALT. Reset -> Start -> instant re-trip, homing never reached,
    // and the only way out was for the operator to jog clear by hand from the manual page.
    //
    // Safe because all three states command NO axis motion: STARTING closes contactors and picks
    // the next state, RECIPE_LOAD runs READ_DBL, PRE_SCAN walks the recipe array. There is
    // nothing for an MC_Halt to halt. The first state that does move -- HOMING(15),
    // PRE_HOME_CLR(13) or POST_HOME_CLR(16) -- was already on this list.
    IF #State <> STATE_HOMING AND #State <> STATE_STOP_GOHOME
       AND #State <> STATE_PRE_HOME_CLR AND #State <> STATE_POST_HOME_CLR
       AND #State <> STATE_MANUAL AND #State <> STATE_STOPPED
       AND #State <> STATE_PNP_HALT AND #State <> STATE_ERROR
       AND #State <> STATE_STARTING AND #State <> STATE_RECIPE_LOAD
       AND #State <> STATE_PRE_SCAN THEN
        IF #HW_PNP_X_Min AND NOT #bHaltX_PNP THEN
            #bHaltX_PNP := TRUE;
            #newErrorFlag := TRUE; #newErrorCode := 16#0121;
            "DB_HMI".ErrorDetail    := 'X MIN proximity triggered - press Reset, then Start (homing clears the zone)';
            #State := STATE_PNP_HALT;
        END_IF;
        IF #HW_PNP_X_Max AND NOT #bHaltX_PNP THEN
            #bHaltX_PNP := TRUE;
            #newErrorFlag := TRUE; #newErrorCode := 16#0122;
            "DB_HMI".ErrorDetail    := 'X MAX proximity triggered - press Reset, then Start (homing clears the zone)';
            #State := STATE_PNP_HALT;
        END_IF;
        IF #HW_PNP_Z_Min AND NOT #bHaltZ_PNP THEN
            #bHaltZ_PNP := TRUE;
            #newErrorFlag := TRUE; #newErrorCode := 16#0123;
            "DB_HMI".ErrorDetail    := 'Z MIN proximity triggered - press Reset, then Start (homing clears the zone)';
            #State := STATE_PNP_HALT;
        END_IF;
        IF #HW_PNP_Z_Max AND NOT #bHaltZ_PNP THEN
            #bHaltZ_PNP := TRUE;
            #newErrorFlag := TRUE; #newErrorCode := 16#0124;
            "DB_HMI".ErrorDetail    := 'Z MAX proximity triggered - press Reset, then Start (homing clears the zone)';
            #State := STATE_PNP_HALT;
        END_IF;
    END_IF;
    // Safety clear: halt flags released when we return to idle
    IF #State = STATE_STOPPED THEN
        #bHaltX_PNP := FALSE;
        #bHaltZ_PNP := FALSE;
    END_IF;

    // Input manager
    #fbInputs(HMI_Start := "DB_HMI".Btn_Start, HMI_Stop := "DB_HMI".Btn_Stop,
              HMI_Pause := "DB_HMI".Btn_Pause, HMI_Reset := "DB_HMI".Btn_Reset,
              Panel_Start := #Panel_Start, Panel_Stop := #Panel_Stop,
              Panel_Pause := #Panel_Pause, Panel_Reset := #Panel_Reset,
              Rem_Start := #Rem_Start, Rem_Stop := #Rem_Stop);

